  MoveL 1967 to (59.09, 49.47, 12.6) mm, rotated rx 0 ry 90 rz 0 deg; joints [-9.8, 3.924, 51.005, 168.083, 55.514, -173.186]
  Set speed (120.0 mm/s)
  MoveL 1968 to (58.95, 49.36, 12.6) mm, rotated rx 0 ry 90 rz 0 deg; joints [-9.795, 3.911, 51.041, 168.092, 55.536, -173.195]
  Set speed (1000.0 mm/s)
  MoveL 1969 to (57.64, 48.99, 12.6) mm, rotated rx 0 ry 90 rz 0 deg; joints [-9.785, 3.793, 51.363, 168.132, 55.734, -173.252]
  MoveL 1970 to (53.2, 41.89, 12.6) mm, rotated rx 0 ry 90 rz 0 deg; joints [-9.389, 3.319, 52.664, 168.719, 56.5, -173.717]
  MoveL 1971 to (53.2, 41.89, 13) mm, rotated rx 0 ry 90 rz 0 deg; joints [-9.389, 3.276, 52.71, 168.719, 56.503, -173.718]
  Set speed (60.0 mm/s)
  Call Extruder(1207.537)
  MoveL 1972 to (56.95, 45.64, 13) mm, rotated rx 0 ry 90 rz 0 deg; joints [-9.584, 3.642, 51.705, 168.401, 55.898, -173.435]
  Call Extruder(1207.555)
  MoveL 1973 to (56.95, 45.51, 13) mm, rotated rx 0 ry 90 rz 0 deg; joints [-9.576, 3.64, 51.71, 168.411, 55.9, -173.441]
  Call Extruder(1207.811)
  MoveL 1974 to (58.88, 45.5, 13) mm, rotated rx 0 ry 90 rz 0 deg; joints [-9.555, 3.805, 51.26, 168.396, 55.618, -173.386]
  Call Extruder(1208.395)
  MoveL 1975 to (58.88, 41.12, 13) mm, rotated rx 0 ry 90 rz 0 deg; joints [-9.282, 3.742, 51.43, 168.74, 55.693, -173.597]
  Call Extruder(1211.736)
  MoveL 1976 to (41.12, 58.88, 13) mm, rotated rx 0 ry 90 rz 0 deg; joints [-10.592, 2.551, 54.735, 167.469, 57.91, -173.266]
  Call Extruder(1211.737)
  MoveL 1977 to (41.12, 58.88, 13) mm, rotated rx 0 ry 90 rz 0 deg; joints [-10.592, 2.551, 54.734, 167.469, 57.91, -173.266]
  Call Extruder(1212.594)
  MoveL 1978 to (41.12, 52.43, 13) mm, rotated rx 0 ry 90 rz 0 deg; joints [-10.184, 2.46, 54.992, 167.969, 58.026, -173.561]
  Call Extruder(1213.807)
  MoveL 1979 to (47.56, 58.88, 13) mm, rotated rx 0 ry 90 rz 0 deg; joints [-10.516, 3.06, 53.31, 167.432, 57.008, -173.078]
  Call Extruder(1214.455)
  MoveL 1980 to (52.43, 58.88, 13) mm, rotated rx 0 ry 90 rz 0 deg; joints [-10.46, 3.459, 52.207, 167.398, 56.314, -172.931]
  Call Extruder(1215.450)
  MoveL 1981 to (57.72, 53.59, 13) mm, rotated rx 0 ry 90 rz 0 deg; joints [-10.071, 3.826, 51.203, 167.771, 55.644, -173.027]
  Call Extruder(1215.604)
  MoveL 1982 to (58.88, 53.59, 13) mm, rotated rx 0 ry 90 rz 0 deg; joints [-10.058, 3.926, 50.931, 167.761, 55.474, -172.991]
  Call Extruder(1216.307)
  MoveL 1983 to (58.88, 58.88, 13) mm, rotated rx 0 ry 90 rz 0 deg; joints [-10.386, 4.008, 50.706, 167.345, 55.376, -172.729]
  Call Extruder(1216.308)
  MoveL 1984 to (58.88, 58.88, 13) mm, rotated rx 0 ry 90 rz 0 deg; joints [-10.386, 4.008, 50.706, 167.345, 55.376, -172.729]
  Call Extruder(1219.649)
  MoveL 1985 to (41.12, 41.12, 13) mm, rotated rx 0 ry 90 rz 0 deg; joints [-9.467, 2.31, 55.416, 168.843, 58.217, -174.07]
  Call Extruder(1220.507)
  MoveL 1986 to (41.12, 47.56, 13) mm, rotated rx 0 ry 90 rz 0 deg; joints [-9.876, 2.394, 55.178, 168.346, 58.11, -173.781]
  Call Extruder(1221.411)
  MoveL 1987 to (45.93, 42.76, 13) mm, rotated rx 0 ry 90 rz 0 deg; joints [-9.52, 2.703, 54.307, 168.694, 57.521, -173.872]
  Call Extruder(1221.446)
  MoveL 1988 to (45.93, 43.02, 13) mm, rotated rx 0 ry 90 rz 0 deg; joints [-9.536, 2.706, 54.297, 168.673, 57.516, -173.86]
  Call Extruder(1221.975)
  MoveL 1989 to (49.9, 43.02, 13) mm, rotated rx 0 ry 90 rz 0 deg; joints [-9.494, 3.023, 53.413, 168.651, 56.955, -173.754]
  Call Extruder(1222.414)
  MoveL 1990 to (53.2, 43.02, 13) mm, rotated rx 0 ry 90 rz 0 deg; joints [-9.46, 3.292, 52.667, 168.631, 56.484, -173.664]
  Call Extruder(1222.667)
  MoveL 1991 to (53.2, 41.12, 13) mm, rotated rx 0 ry 90 rz 0 deg; joints [-9.341, 3.266, 52.739, 168.779, 56.516, -173.754]
  Call Extruder(1223.422)
  MoveL 1992 to (58.88, 41.12, 13) mm, rotated rx 0 ry 90 rz 0 deg; joints [-9.282, 3.742, 51.43, 168.739, 55.693, -173.597]
  MoveL 1993 to (59.08, 41.12, 13) mm, rotated rx 0 ry 90 rz 0 deg; joints [-9.28, 3.76, 51.383, 168.738, 55.663, -173.591]
  Set speed (120.0 mm/s)
  MoveL 1994 to (52.55, 42.37, 13) mm, rotated rx 0 ry 90 rz 0 deg; joints [-9.426, 3.229, 52.84, 168.686, 56.588, -173.713]
  Set speed (1000.0 mm/s)
  MoveL 1995 to (52.48, 42.3, 13) mm, rotated rx 0 ry 90 rz 0 deg; joints [-9.422, 3.223, 52.858, 168.692, 56.599, -173.718]
  Set speed (30.0 mm/s)
  Call Extruder(1223.475)
  MoveL 1996 to (52.48, 41.9, 13) mm, rotated rx 0 ry 90 rz 0 deg; joints [-9.397, 3.217, 52.873, 168.723, 56.606, -173.737]
  Call Extruder(1223.621)
  MoveL 1997 to (52.48, 40.8, 13) mm, rotated rx 0 ry 90 rz 0 deg; joints [-9.328, 3.202, 52.914, 168.808, 56.624, -173.788]
  Call Extruder(1223.675)
  MoveL 1998 to (52.48, 40.4, 13) mm, rotated rx 0 ry 90 rz 0 deg; joints [-9.303, 3.197, 52.929, 168.839, 56.631, -173.807]
  Call Extruder(1223.709)
  MoveL 1999 to (52.88, 40.4, 13) mm, rotated rx 0 ry 90 rz 0 deg; joints [-9.299, 3.23, 52.839, 168.837, 56.573, -173.796]
  Call Extruder(1224.603)
  MoveL 2000 to (59.6, 40.4, 13) mm, rotated rx 0 ry 90 rz 0 deg; joints [-9.23, 3.794, 51.289, 168.79, 55.599, -173.611]
  Call Extruder(1225.378)
  MoveL 2001 to (59.6, 46.22, 13) mm, rotated rx 0 ry 90 rz 0 deg; joints [-9.593, 3.877, 51.062, 168.334, 55.5, -173.33]
  Call Extruder(1225.634)
  MoveL 2002 to (57.67, 46.22, 13) mm, rotated rx 0 ry 90 rz 0 deg; joints [-9.613, 3.712, 51.514, 168.349, 55.782, -173.386]
  Call Extruder(1225.914)
  MoveL 2003 to (57.67, 48.32, 13) mm, rotated rx 0 ry 90 rz 0 deg; joints [-9.744, 3.742, 51.43, 168.184, 55.746, -173.284]
  Call Extruder(1225.967)
  MoveL 2004 to (57.67, 48.72, 13) mm, rotated rx 0 ry 90 rz 0 deg; joints [-9.769, 3.748, 51.414, 168.153, 55.739, -173.265]
  Call Extruder(1226.001)
  MoveL 2005 to (58.07, 48.72, 13) mm, rotated rx 0 ry 90 rz 0 deg; joints [-9.765, 3.782, 51.321, 168.15, 55.68, -173.253]
  Call Extruder(1226.152)
  MoveL 2006 to (59.2, 48.72, 13) mm, rotated rx 0 ry 90 rz 0 deg; joints [-9.752, 3.88, 51.056, 168.141, 55.514, -173.22]
  Call Extruder(1226.205)
  MoveL 2007 to (59.6, 48.72, 13) mm, rotated rx 0 ry 90 rz 0 deg; joints [-9.748, 3.914, 50.962, 168.138, 55.456, -173.208]
  Call Extruder(1226.239)
  MoveL 2008 to (59.6, 49.12, 13) mm, rotated rx 0 ry 90 rz 0 deg; joints [-9.773, 3.92, 50.945, 168.106, 55.449, -173.188]
  Call Extruder(1226.354)
  MoveL 2009 to (59.6, 49.99, 13) mm, rotated rx 0 ry 90 rz 0 deg; joints [-9.827, 3.933, 50.91, 168.038, 55.433, -173.146]
  Call Extruder(1226.407)
  MoveL 2010 to (59.6, 50.39, 13) mm, rotated rx 0 ry 90 rz 0 deg; joints [-9.852, 3.939, 50.894, 168.007, 55.426, -173.126]
  Call Extruder(1226.442)
  MoveL 2011 to (59.2, 50.39, 13) mm, rotated rx 0 ry 90 rz 0 deg; joints [-9.856, 3.904, 50.988, 168.01, 55.485, -173.138]
  Call Extruder(1226.592)
  MoveL 2012 to (58.07, 50.38, 13) mm, rotated rx 0 ry 90 rz 0 deg; joints [-9.868, 3.807, 51.254, 168.02, 55.651, -173.173]
  Call Extruder(1226.646)
  MoveL 2013 to (57.67, 50.38, 13) mm, rotated rx 0 ry 90 rz 0 deg; joints [-9.872, 3.772, 51.348, 168.023, 55.709, -173.185]
  Call Extruder(1226.680)
  MoveL 2014 to (57.67, 50.78, 13) mm, rotated rx 0 ry 90 rz 0 deg; joints [-9.897, 3.778, 51.331, 167.992, 55.702, -173.165]
  Call Extruder(1226.958)
  MoveL 2015 to (57.67, 52.87, 13) mm, rotated rx 0 ry 90 rz 0 deg; joints [-10.027, 3.81, 51.246, 167.828, 55.665, -173.063]
  Call Extruder(1227.215)
  MoveL 2016 to (59.6, 52.87, 13) mm, rotated rx 0 ry 90 rz 0 deg; joints [-10.006, 3.977, 50.791, 167.811, 55.381, -173.004]
  Call Extruder(1228.110)
  MoveL 2017 to (59.6, 59.6, 13) mm, rotated rx 0 ry 90 rz 0 deg; joints [-10.423, 4.083, 50.504, 167.281, 55.256, -172.67]
  Call Extruder(1230.664)
  MoveL 2018 to (40.4, 59.6, 13) mm, rotated rx 0 ry 90 rz 0 deg; joints [-10.646, 2.506, 54.862, 167.417, 57.997, -173.254]
  Call Extruder(1233.218)
  MoveL 2019 to (40.4, 40.4, 13) mm, rotated rx 0 ry 90 rz 0 deg; joints [-9.429, 2.246, 55.596, 168.902, 58.328, -174.12]
  Call Extruder(1234.050)
  MoveL 2020 to (46.65, 40.4, 13) mm, rotated rx 0 ry 90 rz 0 deg; joints [-9.363, 2.728, 54.235, 168.873, 57.458, -173.961]
  Call Extruder(1234.302)
  MoveL 2021 to (46.65, 42.3, 13) mm, rotated rx 0 ry 90 rz 0 deg; joints [-9.483, 2.753, 54.165, 168.725, 57.427, -173.874]
  Call Extruder(1234.629)
  MoveL 2022 to (49.11, 42.3, 13) mm, rotated rx 0 ry 90 rz 0 deg; joints [-9.457, 2.949, 53.619, 168.712, 57.08, -173.809]
  Call Extruder(1234.882)
  MoveL 2023 to (49.11, 40.4, 13) mm, rotated rx 0 ry 90 rz 0 deg; joints [-9.338, 2.924, 53.689, 168.859, 57.111, -173.896]
  Call Extruder(1235.009)
  MoveL 2024 to (50.06, 40.4, 13) mm, rotated rx 0 ry 90 rz 0 deg; joints [-9.328, 3, 53.476, 168.854, 56.976, -173.871]
  Call Extruder(1235.262)
  MoveL 2025 to (50.06, 42.3, 13) mm, rotated rx 0 ry 90 rz 0 deg; joints [-9.447, 3.026, 53.405, 168.706, 56.945, -173.783]
  Call Extruder(1235.531)
  MoveL 2026 to (52.08, 42.3, 13) mm, rotated rx 0 ry 90 rz 0 deg; joints [-9.426, 3.19, 52.949, 168.694, 56.656, -173.729]
  Call Extruder(1235.565)
  MoveL 2027 to (52.48, 42.3, 13) mm, rotated rx 0 ry 90 rz 0 deg; joints [-9.422, 3.223, 52.858, 168.692, 56.599, -173.718]
  Set speed (120.0 mm/s)
  MoveL 2028 to (52.48, 41.9, 13) mm, rotated rx 0 ry 90 rz 0 deg; joints [-9.397, 3.217, 52.873, 168.723, 56.606, -173.737]
  Set speed (1000.0 mm/s)
  MoveL 2029 to (52.58, 41.9, 13) mm, rotated rx 0 ry 90 rz 0 deg; joints [-9.396, 3.226, 52.85, 168.722, 56.591, -173.734]
  MoveL 2030 to (50.03, 42.33, 13) mm, rotated rx 0 ry 90 rz 0 deg; joints [-9.449, 3.024, 53.41, 168.704, 56.948, -173.783]
  MoveL 2031 to (49.58, 42.06, 13) mm, rotated rx 0 ry 90 rz 0 deg; joints [-9.437, 2.984, 53.521, 168.728, 57.017, -173.807]
  Set speed (30.0 mm/s)
  Call Extruder(1235.585)
  MoveL 2032 to (49.58, 42.62, 13) mm, rotated rx 0 ry 90 rz 0 deg; joints [-9.473, 2.991, 53.5, 168.684, 57.007, -173.781]
  Call Extruder(1235.645)
  MoveL 2033 to (49.58, 40.93, 13) mm, rotated rx 0 ry 90 rz 0 deg; joints [-9.366, 2.969, 53.563, 168.816, 57.036, -173.86]
  Set speed (120.0 mm/s)
  MoveL 2034 to (49.91, 40.82, 13) mm, rotated rx 0 ry 90 rz 0 deg; joints [-9.356, 2.994, 53.494, 168.822, 56.991, -173.856]
  Set speed (1000.0 mm/s)
  MoveL 2035 to (50.03, 42.33, 13) mm, rotated rx 0 ry 90 rz 0 deg; joints [-9.449, 3.024, 53.41, 168.704, 56.948, -173.783]
  MoveL 2036 to (52.51, 42.33, 13) mm, rotated rx 0 ry 90 rz 0 deg; joints [-9.423, 3.225, 52.851, 168.689, 56.595, -173.716]
  MoveL 2037 to (53.46, 42.14, 13) mm, rotated rx 0 ry 90 rz 0 deg; joints [-9.402, 3.301, 52.642, 168.697, 56.462, -173.699]
  MoveL 2038 to (53.46, 42.14, 13.4) mm, rotated rx 0 ry 90 rz 0 deg; joints [-9.402, 3.258, 52.689, 168.698, 56.465, -173.699]
  Set speed (60.0 mm/s)
  Call Extruder(1236.301)
  MoveL 2039 to (56.95, 45.64, 13.4) mm, rotated rx 0 ry 90 rz 0 deg; joints [-9.584, 3.599, 51.752, 168.401, 55.901, -173.436]
  Call Extruder(1236.350)
  MoveL 2040 to (56.95, 45.27, 13.4) mm, rotated rx 0 ry 90 rz 0 deg; joints [-9.561, 3.593, 51.766, 168.43, 55.908, -173.454]
  Call Extruder(1236.607)
  MoveL 2041 to (58.88, 45.27, 13.4) mm, rotated rx 0 ry 90 rz 0 deg; joints [-9.541, 3.758, 51.316, 168.415, 55.626, -173.398]
  Call Extruder(1237.159)
  MoveL 2042 to (58.88, 41.12, 13.4) mm, rotated rx 0 ry 90 rz 0 deg; joints [-9.282, 3.699, 51.477, 168.74, 55.697, -173.598]
  Call Extruder(1240.500)
  MoveL 2043 to (41.12, 58.88, 13.4) mm, rotated rx 0 ry 90 rz 0 deg; joints [-10.592, 2.508, 54.78, 167.47, 57.913, -173.267]
  Call Extruder(1240.500)
  MoveL 2044 to (41.12, 58.88, 13.4) mm, rotated rx 0 ry 90 rz 0 deg; joints [-10.592, 2.508, 54.779, 167.47, 57.913, -173.267]
  Call Extruder(1241.358)
  MoveL 2045 to (41.12, 52.43, 13.4) mm, rotated rx 0 ry 90 rz 0 deg; joints [-10.184, 2.417, 55.036, 167.969, 58.028, -173.562]
  Call Extruder(1242.571)
  MoveL 2046 to (47.57, 58.88, 13.4) mm, rotated rx 0 ry 90 rz 0 deg; joints [-10.516, 3.017, 53.356, 167.432, 57.011, -173.079]
  Call Extruder(1243.219)
  MoveL 2047 to (52.43, 58.88, 13.4) mm, rotated rx 0 ry 90 rz 0 deg; joints [-10.46, 3.416, 52.253, 167.398, 56.317, -172.932]
  Call Extruder(1244.171)
  MoveL 2048 to (57.5, 53.82, 13.4) mm, rotated rx 0 ry 90 rz 0 deg; joints [-10.088, 3.766, 51.294, 167.755, 55.677, -173.023]
  Call Extruder(1244.355)
  MoveL 2049 to (58.88, 53.82, 13.4) mm, rotated rx 0 ry 90 rz 0 deg; joints [-10.073, 3.886, 50.969, 167.744, 55.474, -172.981]
  Call Extruder(1245.028)
  MoveL 2050 to (58.88, 58.88, 13.4) mm, rotated rx 0 ry 90 rz 0 deg; joints [-10.386, 3.965, 50.753, 167.345, 55.38, -172.731]
  Call Extruder(1245.029)
  MoveL 2051 to (58.88, 58.88, 13.4) mm, rotated rx 0 ry 90 rz 0 deg; joints [-10.386, 3.965, 50.754, 167.345, 55.38, -172.731]
  Call Extruder(1248.370)
  MoveL 2052 to (41.12, 41.12, 13.4) mm, rotated rx 0 ry 90 rz 0 deg; joints [-9.467, 2.268, 55.46, 168.844, 58.219, -174.07]
  Call Extruder(1249.228)
  MoveL 2053 to (41.12, 47.56, 13.4) mm, rotated rx 0 ry 90 rz 0 deg; joints [-9.876, 2.351, 55.223, 168.346, 58.112, -173.782]
  Call Extruder(1250.090)
  MoveL 2054 to (45.7, 42.98, 13.4) mm, rotated rx 0 ry 90 rz 0 deg; joints [-9.536, 2.645, 54.394, 168.678, 57.551, -173.868]
  Call Extruder(1250.095)
  MoveL 2055 to (45.7, 43.02, 13.4) mm, rotated rx 0 ry 90 rz 0 deg; joints [-9.539, 2.646, 54.392, 168.675, 57.55, -173.867]
  Call Extruder(1250.624)
  MoveL 2056 to (49.68, 43.02, 13.4) mm, rotated rx 0 ry 90 rz 0 deg; joints [-9.497, 2.962, 53.509, 168.653, 56.99, -173.761]
  Call Extruder(1251.127)
  MoveL 2057 to (53.46, 43.02, 13.4) mm, rotated rx 0 ry 90 rz 0 deg; joints [-9.457, 3.27, 52.655, 168.63, 56.45, -173.658]
  Call Extruder(1251.380)
  MoveL 2058 to (53.46, 41.12, 13.4) mm, rotated rx 0 ry 90 rz 0 deg; joints [-9.338, 3.244, 52.727, 168.778, 56.482, -173.747]
  Call Extruder(1252.101)
  MoveL 2059 to (58.88, 41.12, 13.4) mm, rotated rx 0 ry 90 rz 0 deg; joints [-9.282, 3.699, 51.477, 168.74, 55.696, -173.598]
  MoveL 2060 to (59.08, 41.12, 13.4) mm, rotated rx 0 ry 90 rz 0 deg; joints [-9.28, 3.716, 51.43, 168.738, 55.667, -173.592]
  Set speed (120.0 mm/s)
  MoveL 2061 to (52.81, 42.37, 13.4) mm, rotated rx 0 ry 90 rz 0 deg; joints [-9.423, 3.208, 52.828, 168.684, 56.554, -173.707]
  Set speed (1000.0 mm/s)
  MoveL 2062 to (52.74, 42.3, 13.4) mm, rotated rx 0 ry 90 rz 0 deg; joints [-9.419, 3.201, 52.846, 168.69, 56.566, -173.712]
  Set speed (30.0 mm/s)
  Call Extruder(1252.154)
  MoveL 2063 to (52.74, 41.9, 13.4) mm, rotated rx 0 ry 90 rz 0 deg; joints [-9.394, 3.196, 52.861, 168.721, 56.572, -173.73]
  Call Extruder(1252.301)
  MoveL 2064 to (52.74, 40.8, 13.4) mm, rotated rx 0 ry 90 rz 0 deg; joints [-9.325, 3.181, 52.902, 168.807, 56.591, -173.782]
  Call Extruder(1252.354)
  MoveL 2065 to (52.74, 40.4, 13.4) mm, rotated rx 0 ry 90 rz 0 deg; joints [-9.3, 3.175, 52.917, 168.838, 56.597, -173.801]
  Call Extruder(1252.388)
  MoveL 2066 to (53.14, 40.4, 13.4) mm, rotated rx 0 ry 90 rz 0 deg; joints [-9.296, 3.208, 52.827, 168.836, 56.54, -173.79]
  Call Extruder(1253.248)
  MoveL 2067 to (59.6, 40.4, 13.4) mm, rotated rx 0 ry 90 rz 0 deg; joints [-9.23, 3.751, 51.336, 168.791, 55.603, -173.612]
  Call Extruder(1253.991)
  MoveL 2068 to (59.6, 45.98, 13.4) mm, rotated rx 0 ry 90 rz 0 deg; joints [-9.578, 3.83, 51.119, 168.353, 55.508, -173.342]
  Call Extruder(1254.248)
  MoveL 2069 to (57.67, 45.99, 13.4) mm, rotated rx 0 ry 90 rz 0 deg; joints [-9.598, 3.665, 51.57, 168.368, 55.79, -173.398]
  Call Extruder(1254.581)
  MoveL 2070 to (57.67, 48.49, 13.4) mm, rotated rx 0 ry 90 rz 0 deg; joints [-9.754, 3.701, 51.471, 168.172, 55.747, -173.277]
  Call Extruder(1254.837)
  MoveL 2071 to (59.6, 48.49, 13.4) mm, rotated rx 0 ry 90 rz 0 deg; joints [-9.734, 3.867, 51.019, 168.157, 55.464, -173.22]
  Call Extruder(1255.066)
  MoveL 2072 to (59.6, 50.21, 13.4) mm, rotated rx 0 ry 90 rz 0 deg; joints [-9.84, 3.893, 50.949, 168.022, 55.433, -173.136]
  Call Extruder(1255.119)
  MoveL 2073 to (59.6, 50.61, 13.4) mm, rotated rx 0 ry 90 rz 0 deg; joints [-9.865, 3.899, 50.932, 167.99, 55.426, -173.116]
  Call Extruder(1255.154)
  MoveL 2074 to (59.2, 50.61, 13.4) mm, rotated rx 0 ry 90 rz 0 deg; joints [-9.87, 3.864, 51.027, 167.993, 55.485, -173.129]
  Call Extruder(1255.304)
  MoveL 2075 to (58.07, 50.61, 13.4) mm, rotated rx 0 ry 90 rz 0 deg; joints [-9.882, 3.767, 51.292, 168.003, 55.651, -173.163]
  Call Extruder(1255.358)
  MoveL 2076 to (57.67, 50.61, 13.4) mm, rotated rx 0 ry 90 rz 0 deg; joints [-9.886, 3.733, 51.386, 168.006, 55.709, -173.175]
  Call Extruder(1255.392)
  MoveL 2077 to (57.67, 51.01, 13.4) mm, rotated rx 0 ry 90 rz 0 deg; joints [-9.911, 3.738, 51.37, 167.975, 55.702, -173.155]
  Call Extruder(1255.670)
  MoveL 2078 to (57.67, 53.1, 13.4) mm, rotated rx 0 ry 90 rz 0 deg; joints [-10.041, 3.77, 51.284, 167.811, 55.665, -173.053]
  Call Extruder(1255.927)
  MoveL 2079 to (59.6, 53.1, 13.4) mm, rotated rx 0 ry 90 rz 0 deg; joints [-10.02, 3.937, 50.829, 167.794, 55.381, -172.994]
  Call Extruder(1256.792)
  MoveL 2080 to (59.6, 59.6, 13.4) mm, rotated rx 0 ry 90 rz 0 deg; joints [-10.423, 4.039, 50.552, 167.282, 55.26, -172.672]
  Call Extruder(1259.347)
  MoveL 2081 to (40.4, 59.6, 13.4) mm, rotated rx 0 ry 90 rz 0 deg; joints [-10.646, 2.463, 54.906, 167.418, 57.999, -173.254]
  Call Extruder(1261.901)
  MoveL 2082 to (40.4, 40.4, 13.4) mm, rotated rx 0 ry 90 rz 0 deg; joints [-9.429, 2.204, 55.641, 168.902, 58.33, -174.12]
  Call Extruder(1262.702)
  MoveL 2083 to (46.42, 40.4, 13.4) mm, rotated rx 0 ry 90 rz 0 deg; joints [-9.366, 2.668, 54.33, 168.874, 57.493, -173.967]
  Call Extruder(1262.955)
  MoveL 2084 to (46.42, 42.3, 13.4) mm, rotated rx 0 ry 90 rz 0 deg; joints [-9.486, 2.693, 54.26, 168.727, 57.461, -173.88]
  Call Extruder(1263.282)
  MoveL 2085 to (48.88, 42.3, 13.4) mm, rotated rx 0 ry 90 rz 0 deg; joints [-9.46, 2.888, 53.715, 168.713, 57.115, -173.816]
  Call Extruder(1263.535)
  MoveL 2086 to (48.88, 40.4, 13.4) mm, rotated rx 0 ry 90 rz 0 deg; joints [-9.34, 2.863, 53.785, 168.861, 57.146, -173.903]
  Call Extruder(1263.725)
  MoveL 2087 to (50.31, 40.4, 13.4) mm, rotated rx 0 ry 90 rz 0 deg; joints [-9.325, 2.978, 53.465, 168.853, 56.943, -173.865]
  Call Extruder(1263.978)
  MoveL 2088 to (50.31, 42.3, 13.4) mm, rotated rx 0 ry 90 rz 0 deg; joints [-9.445, 3.003, 53.394, 168.705, 56.912, -173.777]
  Call Extruder(1264.248)
  MoveL 2089 to (52.34, 42.3, 13.4) mm, rotated rx 0 ry 90 rz 0 deg; joints [-9.424, 3.168, 52.937, 168.693, 56.623, -173.723]
  Call Extruder(1264.282)
  MoveL 2090 to (52.74, 42.3, 13.4) mm, rotated rx 0 ry 90 rz 0 deg; joints [-9.419, 3.201, 52.846, 168.69, 56.566, -173.712]
  Set speed (120.0 mm/s)
  MoveL 2091 to (52.74, 41.9, 13.4) mm, rotated rx 0 ry 90 rz 0 deg; joints [-9.394, 3.196, 52.861, 168.721, 56.572, -173.73]
  Set speed (1000.0 mm/s)
  MoveL 2092 to (52.84, 41.9, 13.4) mm, rotated rx 0 ry 90 rz 0 deg; joints [-9.393, 3.204, 52.838, 168.721, 56.558, -173.728]
  MoveL 2093 to (50.28, 42.33, 13.4) mm, rotated rx 0 ry 90 rz 0 deg; joints [-9.447, 3.001, 53.399, 168.703, 56.915, -173.777]
  MoveL 2094 to (49.6, 41.68, 13.4) mm, rotated rx 0 ry 90 rz 0 deg; joints [-9.413, 2.937, 53.578, 168.758, 57.024, -173.825]
  Set speed (30.0 mm/s)
  Call Extruder(1264.377)
  MoveL 2095 to (49.6, 41.11, 13.4) mm, rotated rx 0 ry 90 rz 0 deg; joints [-9.377, 2.93, 53.598, 168.802, 57.033, -173.851]
  Call Extruder(1264.444)
  MoveL 2096 to (49.88, 40.83, 13.4) mm, rotated rx 0 ry 90 rz 0 deg; joints [-9.357, 2.949, 53.546, 168.822, 56.998, -173.857]
  Set speed (120.0 mm/s)
  MoveL 2097 to (49.83, 40.78, 13.4) mm, rotated rx 0 ry 90 rz 0 deg; joints [-9.354, 2.944, 53.56, 168.826, 57.006, -173.861]
  Set speed (1000.0 mm/s)
  MoveL 2098 to (49.25, 41.9, 13.4) mm, rotated rx 0 ry 90 rz 0 deg; joints [-9.431, 2.913, 53.646, 168.742, 57.069, -173.824]
  Set speed (30.0 mm/s)
  Call Extruder(1264.508)
  MoveL 2099 to (49.94, 42.58, 13.4) mm, rotated rx 0 ry 90 rz 0 deg; joints [-9.466, 2.977, 53.468, 168.685, 56.961, -173.774]
  Set speed (120.0 mm/s)
  MoveL 2100 to (49.53, 42.74, 13.4) mm, rotated rx 0 ry 90 rz 0 deg; joints [-9.481, 2.946, 53.554, 168.676, 57.016, -173.778]
  Set speed (30.0 mm/s)
  Call Extruder(1264.534)
  MoveL 2101 to (49.25, 42.47, 13.4) mm, rotated rx 0 ry 90 rz 0 deg; joints [-9.466, 2.92, 53.625, 168.699, 57.059, -173.798]
  Set speed (120.0 mm/s)
  MoveL 2102 to (49.45, 42.87, 13.4) mm, rotated rx 0 ry 90 rz 0 deg; joints [-9.489, 2.941, 53.568, 168.666, 57.026, -173.774]
  Set speed (1000.0 mm/s)
  MoveL 2103 to (46.97, 42.43, 13.4) mm, rotated rx 0 ry 90 rz 0 deg; joints [-9.488, 2.738, 54.133, 168.714, 57.382, -173.86]
  MoveL 2104 to (41.12, 41.12, 13.4) mm, rotated rx 0 ry 90 rz 0 deg; joints [-9.467, 2.268, 55.46, 168.844, 58.219, -174.07]
  MoveL 2105 to (41.12, 41.12, 13.8) mm, rotated rx 0 ry 90 rz 0 deg; joints [-9.467, 2.225, 55.505, 168.844, 58.221, -174.071]
  Set speed (60.0 mm/s)
  Call Extruder(1267.875)
  MoveL 2106 to (58.88, 58.88, 13.8) mm, rotated rx 0 ry 90 rz 0 deg; joints [-10.386, 3.921, 50.801, 167.346, 55.384, -172.732]
  Call Extruder(1268.733)
  MoveL 2107 to (52.43, 58.88, 13.8) mm, rotated rx 0 ry 90 rz 0 deg; joints [-10.46, 3.373, 52.3, 167.399, 56.32, -172.933]
  Call Extruder(1269.643)
  MoveL 2108 to (57.27, 54.04, 13.8) mm, rotated rx 0 ry 90 rz 0 deg; joints [-10.104, 3.707, 51.385, 167.74, 55.709, -173.02]
  Call Extruder(1269.686)
  MoveL 2109 to (56.95, 54.04, 13.8) mm, rotated rx 0 ry 90 rz 0 deg; joints [-10.108, 3.679, 51.46, 167.743, 55.756, -173.03]
  Call Extruder(1270.209)
  MoveL 2110 to (56.95, 50.11, 13.8) mm, rotated rx 0 ry 90 rz 0 deg; joints [-9.863, 3.621, 51.621, 168.051, 55.827, -173.221]
  Call Extruder(1270.466)
  MoveL 2111 to (58.88, 50.11, 13.8) mm, rotated rx 0 ry 90 rz 0 deg; joints [-9.842, 3.786, 51.169, 168.036, 55.545, -173.164]
  Call Extruder(1270.617)
  MoveL 2112 to (58.88, 48.98, 13.8) mm, rotated rx 0 ry 90 rz 0 deg; joints [-9.772, 3.769, 51.216, 168.125, 55.565, -173.219]
  Call Extruder(1270.874)
  MoveL 2113 to (56.95, 48.98, 13.8) mm, rotated rx 0 ry 90 rz 0 deg; joints [-9.792, 3.604, 51.666, 168.14, 55.847, -173.276]
  Call Extruder(1271.318)
  MoveL 2114 to (56.95, 45.64, 13.8) mm, rotated rx 0 ry 90 rz 0 deg; joints [-9.584, 3.556, 51.798, 168.401, 55.905, -173.437]
  Call Extruder(1271.927)
  MoveL 2115 to (53.72, 42.4, 13.8) mm, rotated rx 0 ry 90 rz 0 deg; joints [-9.416, 3.24, 52.667, 168.677, 56.427, -173.681]
  Call Extruder(1272.097)
  MoveL 2116 to (53.72, 41.12, 13.8) mm, rotated rx 0 ry 90 rz 0 deg; joints [-9.335, 3.222, 52.715, 168.776, 56.449, -173.741]
  Call Extruder(1272.784)
  MoveL 2117 to (58.88, 41.12, 13.8) mm, rotated rx 0 ry 90 rz 0 deg; joints [-9.282, 3.656, 51.524, 168.74, 55.7, -173.599]
  Call Extruder(1272.784)
  MoveL 2118 to (58.88, 41.12, 13.8) mm, rotated rx 0 ry 90 rz 0 deg; joints [-9.282, 3.656, 51.524, 168.741, 55.7, -173.599]
  Call Extruder(1276.126)
  MoveL 2119 to (41.12, 58.88, 13.8) mm, rotated rx 0 ry 90 rz 0 deg; joints [-10.592, 2.466, 54.824, 167.47, 57.915, -173.267]
  Call Extruder(1276.983)
  MoveL 2120 to (47.56, 58.88, 13.8) mm, rotated rx 0 ry 90 rz 0 deg; joints [-10.516, 2.974, 53.402, 167.432, 57.014, -173.08]
  Call Extruder(1278.196)
  MoveL 2121 to (41.12, 52.43, 13.8) mm, rotated rx 0 ry 90 rz 0 deg; joints [-10.184, 2.375, 55.081, 167.97, 58.03, -173.562]
  Call Extruder(1278.844)
  MoveL 2122 to (41.12, 47.56, 13.8) mm, rotated rx 0 ry 90 rz 0 deg; joints [-9.876, 2.309, 55.267, 168.346, 58.114, -173.782]
  Call Extruder(1279.699)
  MoveL 2123 to (45.66, 43.02, 13.8) mm, rotated rx 0 ry 90 rz 0 deg; joints [-9.539, 2.601, 54.446, 168.675, 57.558, -173.868]
  MoveL 2124 to (45.8, 42.88, 13.8) mm, rotated rx 0 ry 90 rz 0 deg; joints [-9.529, 2.61, 54.42, 168.686, 57.541, -173.871]
  Set speed (120.0 mm/s)
  MoveL 2125 to (48.68, 42.33, 13.8) mm, rotated rx 0 ry 90 rz 0 deg; joints [-9.464, 2.83, 53.803, 168.713, 57.146, -173.82]
  Set speed (1000.0 mm/s)
  MoveL 2126 to (49.85, 41.12, 13.8) mm, rotated rx 0 ry 90 rz 0 deg; joints [-9.375, 2.907, 53.589, 168.8, 57.001, -173.845]
  Set speed (60.0 mm/s)
  Call Extruder(1279.761)
  MoveL 2127 to (49.37, 41.12, 13.8) mm, rotated rx 0 ry 90 rz 0 deg; joints [-9.38, 2.869, 53.694, 168.803, 57.067, -173.857]
  Call Extruder(1280.014)
  MoveL 2128 to (49.37, 43.02, 13.8) mm, rotated rx 0 ry 90 rz 0 deg; joints [-9.5, 2.895, 53.623, 168.655, 57.036, -173.77]
  Call Extruder(1280.533)
  MoveL 2129 to (45.48, 43.02, 13.8) mm, rotated rx 0 ry 90 rz 0 deg; joints [-9.541, 2.586, 54.487, 168.676, 57.584, -173.873]
  Call Extruder(1280.785)
  MoveL 2130 to (45.48, 41.12, 13.8) mm, rotated rx 0 ry 90 rz 0 deg; joints [-9.421, 2.561, 54.556, 168.824, 57.616, -173.959]
  Call Extruder(1281.365)
  MoveL 2131 to (41.12, 41.12, 13.8) mm, rotated rx 0 ry 90 rz 0 deg; joints [-9.467, 2.225, 55.504, 168.844, 58.221, -174.071]
  Call Extruder(1281.366)
  MoveL 2132 to (41.12, 41.12, 13.8) mm, rotated rx 0 ry 90 rz 0 deg; joints [-9.467, 2.225, 55.505, 168.844, 58.221, -174.071]
  Set speed (120.0 mm/s)
  MoveL 2133 to (46.17, 42.33, 13.8) mm, rotated rx 0 ry 90 rz 0 deg; joints [-9.49, 2.631, 54.36, 168.726, 57.499, -173.886]
  Set speed (1000.0 mm/s)
  MoveL 2134 to (53.07, 42.37, 13.8) mm, rotated rx 0 ry 90 rz 0 deg; joints [-9.42, 3.186, 52.816, 168.683, 56.521, -173.7]
  MoveL 2135 to (53, 42.3, 13.8) mm, rotated rx 0 ry 90 rz 0 deg; joints [-9.417, 3.179, 52.834, 168.689, 56.532, -173.706]
  Set speed (30.0 mm/s)
  Call Extruder(1281.419)
  MoveL 2136 to (53, 41.9, 13.8) mm, rotated rx 0 ry 90 rz 0 deg; joints [-9.392, 3.174, 52.849, 168.72, 56.539, -173.724]
  Call Extruder(1281.565)
  MoveL 2137 to (52.99, 40.8, 13.8) mm, rotated rx 0 ry 90 rz 0 deg; joints [-9.323, 3.159, 52.891, 168.806, 56.557, -173.776]
  Call Extruder(1281.618)
  MoveL 2138 to (52.99, 40.4, 13.8) mm, rotated rx 0 ry 90 rz 0 deg; joints [-9.297, 3.153, 52.906, 168.837, 56.564, -173.794]
  Call Extruder(1281.653)
  MoveL 2139 to (53.39, 40.4, 13.8) mm, rotated rx 0 ry 90 rz 0 deg; joints [-9.293, 3.186, 52.815, 168.834, 56.507, -173.784]
  Call Extruder(1282.478)
  MoveL 2140 to (59.6, 40.4, 13.8) mm, rotated rx 0 ry 90 rz 0 deg; joints [-9.23, 3.708, 51.383, 168.791, 55.607, -173.613]
  Call Extruder(1283.190)
  MoveL 2141 to (59.6, 45.75, 13.8) mm, rotated rx 0 ry 90 rz 0 deg; joints [-9.563, 3.784, 51.176, 168.373, 55.516, -173.355]
  Call Extruder(1283.446)
  MoveL 2142 to (57.67, 45.75, 13.8) mm, rotated rx 0 ry 90 rz 0 deg; joints [-9.583, 3.618, 51.627, 168.387, 55.798, -173.411]
  Call Extruder(1283.780)
  MoveL 2143 to (57.67, 48.26, 13.8) mm, rotated rx 0 ry 90 rz 0 deg; joints [-9.74, 3.655, 51.527, 168.191, 55.754, -173.29]
  Call Extruder(1284.037)
  MoveL 2144 to (59.6, 48.26, 13.8) mm, rotated rx 0 ry 90 rz 0 deg; joints [-9.719, 3.82, 51.075, 168.176, 55.472, -173.233]
  Call Extruder(1284.326)
  MoveL 2145 to (59.6, 50.43, 13.8) mm, rotated rx 0 ry 90 rz 0 deg; joints [-9.854, 3.853, 50.987, 168.005, 55.433, -173.126]
  Call Extruder(1284.379)
  MoveL 2146 to (59.6, 50.83, 13.8) mm, rotated rx 0 ry 90 rz 0 deg; joints [-9.879, 3.859, 50.971, 167.973, 55.426, -173.107]
  Call Extruder(1284.414)
  MoveL 2147 to (59.2, 50.83, 13.8) mm, rotated rx 0 ry 90 rz 0 deg; joints [-9.883, 3.824, 51.065, 167.977, 55.485, -173.119]
  Call Extruder(1284.564)
  MoveL 2148 to (58.07, 50.83, 13.8) mm, rotated rx 0 ry 90 rz 0 deg; joints [-9.896, 3.727, 51.33, 167.986, 55.651, -173.153]
  Call Extruder(1284.617)
  MoveL 2149 to (57.67, 50.83, 13.8) mm, rotated rx 0 ry 90 rz 0 deg; joints [-9.9, 3.693, 51.424, 167.989, 55.709, -173.165]
  Call Extruder(1284.652)
  MoveL 2150 to (57.67, 51.23, 13.8) mm, rotated rx 0 ry 90 rz 0 deg; joints [-9.925, 3.699, 51.407, 167.958, 55.702, -173.145]
  Call Extruder(1284.930)
  MoveL 2151 to (57.67, 53.32, 13.8) mm, rotated rx 0 ry 90 rz 0 deg; joints [-10.055, 3.73, 51.321, 167.793, 55.664, -173.043]
  Call Extruder(1285.187)
  MoveL 2152 to (59.6, 53.33, 13.8) mm, rotated rx 0 ry 90 rz 0 deg; joints [-10.034, 3.897, 50.867, 167.777, 55.381, -172.984]
  Call Extruder(1286.022)
  MoveL 2153 to (59.6, 59.6, 13.8) mm, rotated rx 0 ry 90 rz 0 deg; joints [-10.423, 3.996, 50.599, 167.283, 55.264, -172.673]
  Call Extruder(1288.576)
  MoveL 2154 to (40.4, 59.6, 13.8) mm, rotated rx 0 ry 90 rz 0 deg; joints [-10.646, 2.421, 54.951, 167.418, 58.001, -173.255]
  Call Extruder(1291.131)
  MoveL 2155 to (40.4, 40.4, 13.8) mm, rotated rx 0 ry 90 rz 0 deg; joints [-9.429, 2.162, 55.685, 168.902, 58.332, -174.121]
  Call Extruder(1291.849)
  MoveL 2156 to (45.8, 40.4, 13.8) mm, rotated rx 0 ry 90 rz 0 deg; joints [-9.372, 2.577, 54.512, 168.878, 57.583, -173.984]
  Call Extruder(1291.902)
  MoveL 2157 to (46.2, 40.4, 13.8) mm, rotated rx 0 ry 90 rz 0 deg; joints [-9.368, 2.608, 54.424, 168.876, 57.527, -173.973]
  Call Extruder(1291.937)
  MoveL 2158 to (46.2, 40.8, 13.8) mm, rotated rx 0 ry 90 rz 0 deg; joints [-9.393, 2.613, 54.41, 168.845, 57.52, -173.955]
  Call Extruder(1292.083)
  MoveL 2159 to (46.2, 41.9, 13.8) mm, rotated rx 0 ry 90 rz 0 deg; joints [-9.463, 2.628, 54.37, 168.759, 57.502, -173.905]
  Call Extruder(1292.136)
  MoveL 2160 to (46.2, 42.3, 13.8) mm, rotated rx 0 ry 90 rz 0 deg; joints [-9.488, 2.633, 54.355, 168.728, 57.496, -173.887]
  Call Extruder(1292.171)
  MoveL 2161 to (46.6, 42.3, 13.8) mm, rotated rx 0 ry 90 rz 0 deg; joints [-9.484, 2.664, 54.267, 168.726, 57.439, -173.876]
  Call Extruder(1292.444)
  MoveL 2162 to (48.65, 42.3, 13.8) mm, rotated rx 0 ry 90 rz 0 deg; joints [-9.462, 2.827, 53.811, 168.715, 57.15, -173.822]
  Call Extruder(1292.697)
  MoveL 2163 to (48.66, 40.4, 13.8) mm, rotated rx 0 ry 90 rz 0 deg; joints [-9.342, 2.803, 53.88, 168.863, 57.181, -173.909]
  Call Extruder(1292.951)
  MoveL 2164 to (50.56, 40.4, 13.8) mm, rotated rx 0 ry 90 rz 0 deg; joints [-9.323, 2.956, 53.454, 168.852, 56.911, -173.859]
  Call Extruder(1293.204)
  MoveL 2165 to (50.57, 42.3, 13.8) mm, rotated rx 0 ry 90 rz 0 deg; joints [-9.442, 2.981, 53.383, 168.704, 56.879, -173.771]
  Call Extruder(1293.474)
  MoveL 2166 to (52.6, 42.3, 13.8) mm, rotated rx 0 ry 90 rz 0 deg; joints [-9.421, 3.146, 52.925, 168.692, 56.589, -173.716]
  Call Extruder(1293.508)
  MoveL 2167 to (53, 42.3, 13.8) mm, rotated rx 0 ry 90 rz 0 deg; joints [-9.417, 3.179, 52.834, 168.689, 56.532, -173.706]
  Set speed (120.0 mm/s)
  MoveL 2168 to (53, 41.9, 13.8) mm, rotated rx 0 ry 90 rz 0 deg; joints [-9.392, 3.174, 52.849, 168.72, 56.539, -173.724]
  Set speed (1000.0 mm/s)
  MoveL 2169 to (53.8, 41.9, 13.8) mm, rotated rx 0 ry 90 rz 0 deg; joints [-9.383, 3.24, 52.667, 168.715, 56.424, -173.702]
  MoveL 2170 to (46.17, 42.33, 13.8) mm, rotated rx 0 ry 90 rz 0 deg; joints [-9.49, 2.631, 54.36, 168.726, 57.499, -173.886]
  MoveL 2171 to (41.12, 41.12, 13.8) mm, rotated rx 0 ry 90 rz 0 deg; joints [-9.467, 2.225, 55.505, 168.844, 58.221, -174.071]
  MoveL 2172 to (41.12, 41.12, 14.2) mm, rotated rx 0 ry 90 rz 0 deg; joints [-9.467, 2.183, 55.549, 168.844, 58.224, -174.071]
  Set speed (60.0 mm/s)
  Call Extruder(1296.850)
  MoveL 2173 to (58.88, 58.88, 14.2) mm, rotated rx 0 ry 90 rz 0 deg; joints [-10.386, 3.878, 50.849, 167.347, 55.388, -172.733]
  Call Extruder(1297.707)
  MoveL 2174 to (52.43, 58.88, 14.2) mm, rotated rx 0 ry 90 rz 0 deg; joints [-10.46, 3.33, 52.346, 167.399, 56.324, -172.934]
  Call Extruder(1298.575)
  MoveL 2175 to (57.04, 54.27, 14.2) mm, rotated rx 0 ry 90 rz 0 deg; joints [-10.121, 3.648, 51.475, 167.725, 55.742, -173.017]
  Call Extruder(1298.588)
  MoveL 2176 to (56.95, 54.27, 14.2) mm, rotated rx 0 ry 90 rz 0 deg; joints [-10.122, 3.64, 51.497, 167.726, 55.756, -173.02]
  Call Extruder(1299.112)
  MoveL 2177 to (56.95, 50.33, 14.2) mm, rotated rx 0 ry 90 rz 0 deg; joints [-9.877, 3.581, 51.659, 168.034, 55.827, -173.211]
  Call Extruder(1299.369)
  MoveL 2178 to (58.88, 50.33, 14.2) mm, rotated rx 0 ry 90 rz 0 deg; joints [-9.856, 3.746, 51.208, 168.019, 55.545, -173.154]
  Call Extruder(1299.581)
  MoveL 2179 to (58.88, 48.74, 14.2) mm, rotated rx 0 ry 90 rz 0 deg; joints [-9.757, 3.722, 51.272, 168.144, 55.573, -173.231]
  Call Extruder(1299.837)
  MoveL 2180 to (56.95, 48.74, 14.2) mm, rotated rx 0 ry 90 rz 0 deg; joints [-9.778, 3.558, 51.722, 168.159, 55.854, -173.288]
  Call Extruder(1300.250)
  MoveL 2181 to (56.95, 45.64, 14.2) mm, rotated rx 0 ry 90 rz 0 deg; joints [-9.584, 3.513, 51.845, 168.402, 55.908, -173.438]
  Call Extruder(1300.811)
  MoveL 2182 to (53.97, 42.65, 14.2) mm, rotated rx 0 ry 90 rz 0 deg; joints [-9.429, 3.221, 52.645, 168.656, 56.39, -173.663]
  Call Extruder(1301.015)
  MoveL 2183 to (53.97, 41.12, 14.2) mm, rotated rx 0 ry 90 rz 0 deg; joints [-9.333, 3.2, 52.703, 168.775, 56.415, -173.735]
  Call Extruder(1301.669)
  MoveL 2184 to (58.88, 41.12, 14.2) mm, rotated rx 0 ry 90 rz 0 deg; joints [-9.282, 3.613, 51.571, 168.741, 55.704, -173.6]
  Call Extruder(1301.669)
  MoveL 2185 to (58.88, 41.12, 14.2) mm, rotated rx 0 ry 90 rz 0 deg; joints [-9.282, 3.613, 51.571, 168.741, 55.704, -173.6]
  Call Extruder(1305.010)
  MoveL 2186 to (41.12, 58.88, 14.2) mm, rotated rx 0 ry 90 rz 0 deg; joints [-10.592, 2.424, 54.869, 167.47, 57.917, -173.268]
  Call Extruder(1305.868)
  MoveL 2187 to (47.56, 58.88, 14.2) mm, rotated rx 0 ry 90 rz 0 deg; joints [-10.516, 2.932, 53.448, 167.433, 57.017, -173.08]
  Call Extruder(1307.081)
  MoveL 2188 to (41.12, 52.43, 14.2) mm, rotated rx 0 ry 90 rz 0 deg; joints [-10.184, 2.333, 55.126, 167.97, 58.033, -173.563]
  Call Extruder(1307.728)
  MoveL 2189 to (41.12, 47.57, 14.2) mm, rotated rx 0 ry 90 rz 0 deg; joints [-9.876, 2.267, 55.312, 168.346, 58.116, -173.783]
  Call Extruder(1308.583)
  MoveL 2190 to (45.66, 43.02, 14.2) mm, rotated rx 0 ry 90 rz 0 deg; joints [-9.539, 2.558, 54.491, 168.676, 57.561, -173.869]
  MoveL 2191 to (45.81, 42.88, 14.2) mm, rotated rx 0 ry 90 rz 0 deg; joints [-9.529, 2.567, 54.465, 168.686, 57.544, -173.872]
  Set speed (120.0 mm/s)
  MoveL 2192 to (48.46, 42.33, 14.2) mm, rotated rx 0 ry 90 rz 0 deg; joints [-9.466, 2.769, 53.899, 168.714, 57.18, -173.827]
  Set speed (1000.0 mm/s)
  MoveL 2193 to (50.1, 41.12, 14.2) mm, rotated rx 0 ry 90 rz 0 deg; joints [-9.373, 2.885, 53.577, 168.799, 56.968, -173.839]
  Set speed (60.0 mm/s)
  Call Extruder(1308.710)
  MoveL 2194 to (49.15, 41.12, 14.2) mm, rotated rx 0 ry 90 rz 0 deg; joints [-9.383, 2.809, 53.789, 168.804, 57.102, -173.864]
  Call Extruder(1308.963)
  MoveL 2195 to (49.15, 43.02, 14.2) mm, rotated rx 0 ry 90 rz 0 deg; joints [-9.502, 2.834, 53.719, 168.657, 57.071, -173.777]
  Call Extruder(1309.481)
  MoveL 2196 to (45.25, 43.02, 14.2) mm, rotated rx 0 ry 90 rz 0 deg; joints [-9.544, 2.526, 54.581, 168.678, 57.618, -173.88]
  Call Extruder(1309.734)
  MoveL 2197 to (45.25, 41.12, 14.2) mm, rotated rx 0 ry 90 rz 0 deg; joints [-9.423, 2.501, 54.65, 168.825, 57.65, -173.966]
  Call Extruder(1310.284)
  MoveL 2198 to (41.12, 41.12, 14.2) mm, rotated rx 0 ry 90 rz 0 deg; joints [-9.467, 2.183, 55.549, 168.844, 58.223, -174.071]
  Call Extruder(1310.284)
  MoveL 2199 to (41.12, 41.12, 14.2) mm, rotated rx 0 ry 90 rz 0 deg; joints [-9.467, 2.183, 55.549, 168.844, 58.224, -174.071]
  Set speed (120.0 mm/s)
  MoveL 2200 to (45.94, 42.33, 14.2) mm, rotated rx 0 ry 90 rz 0 deg; joints [-9.492, 2.571, 54.455, 168.728, 57.533, -173.893]
  Set speed (1000.0 mm/s)
  MoveL 2201 to (53.32, 42.37, 14.2) mm, rotated rx 0 ry 90 rz 0 deg; joints [-9.418, 3.164, 52.804, 168.682, 56.488, -173.694]
  MoveL 2202 to (53.25, 42.3, 14.2) mm, rotated rx 0 ry 90 rz 0 deg; joints [-9.414, 3.157, 52.822, 168.688, 56.499, -173.699]
  Set speed (30.0 mm/s)
  Call Extruder(1310.337)
  MoveL 2203 to (53.25, 41.9, 14.2) mm, rotated rx 0 ry 90 rz 0 deg; joints [-9.389, 3.152, 52.837, 168.719, 56.505, -173.718]
  Call Extruder(1310.483)
  MoveL 2204 to (53.25, 40.8, 14.2) mm, rotated rx 0 ry 90 rz 0 deg; joints [-9.32, 3.137, 52.879, 168.805, 56.524, -173.77]
  Call Extruder(1310.536)
  MoveL 2205 to (53.25, 40.4, 14.2) mm, rotated rx 0 ry 90 rz 0 deg; joints [-9.295, 3.131, 52.894, 168.836, 56.53, -173.788]
  Call Extruder(1310.571)
  MoveL 2206 to (53.65, 40.4, 14.2) mm, rotated rx 0 ry 90 rz 0 deg; joints [-9.291, 3.164, 52.803, 168.833, 56.473, -173.778]
  Call Extruder(1311.363)
  MoveL 2207 to (59.6, 40.4, 14.2) mm, rotated rx 0 ry 90 rz 0 deg; joints [-9.23, 3.664, 51.43, 168.792, 55.611, -173.614]
  Call Extruder(1312.042)
  MoveL 2208 to (59.6, 45.51, 14.2) mm, rotated rx 0 ry 90 rz 0 deg; joints [-9.548, 3.737, 51.232, 168.392, 55.524, -173.367]
  Call Extruder(1312.298)
  MoveL 2209 to (57.67, 45.51, 14.2) mm, rotated rx 0 ry 90 rz 0 deg; joints [-9.568, 3.572, 51.683, 168.407, 55.806, -173.423]
  Call Extruder(1312.580)
  MoveL 2210 to (57.67, 47.62, 14.2) mm, rotated rx 0 ry 90 rz 0 deg; joints [-9.7, 3.602, 51.599, 168.241, 55.769, -173.321]
  Call Extruder(1312.633)
  MoveL 2211 to (57.67, 48.02, 14.2) mm, rotated rx 0 ry 90 rz 0 deg; joints [-9.725, 3.608, 51.583, 168.21, 55.762, -173.302]
  Call Extruder(1312.667)
  MoveL 2212 to (58.07, 48.02, 14.2) mm, rotated rx 0 ry 90 rz 0 deg; joints [-9.721, 3.642, 51.49, 168.207, 55.703, -173.29]
  Call Extruder(1312.817)
  MoveL 2213 to (59.2, 48.02, 14.2) mm, rotated rx 0 ry 90 rz 0 deg; joints [-9.709, 3.739, 51.226, 168.198, 55.539, -173.257]
  Call Extruder(1312.870)
  MoveL 2214 to (59.6, 48.02, 14.2) mm, rotated rx 0 ry 90 rz 0 deg; joints [-9.705, 3.774, 51.132, 168.194, 55.48, -173.245]
  Call Extruder(1312.905)
  MoveL 2215 to (59.6, 48.42, 14.2) mm, rotated rx 0 ry 90 rz 0 deg; joints [-9.729, 3.78, 51.116, 168.163, 55.473, -173.226]
  Call Extruder(1313.202)
  MoveL 2216 to (59.6, 50.65, 14.2) mm, rotated rx 0 ry 90 rz 0 deg; joints [-9.868, 3.813, 51.025, 167.988, 55.433, -173.116]
  Call Extruder(1313.255)
  MoveL 2217 to (59.6, 51.05, 14.2) mm, rotated rx 0 ry 90 rz 0 deg; joints [-9.893, 3.819, 51.009, 167.956, 55.426, -173.097]
  Call Extruder(1313.290)
  MoveL 2218 to (59.2, 51.05, 14.2) mm, rotated rx 0 ry 90 rz 0 deg; joints [-9.897, 3.784, 51.103, 167.96, 55.485, -173.109]
  Call Extruder(1313.440)
  MoveL 2219 to (58.07, 51.05, 14.2) mm, rotated rx 0 ry 90 rz 0 deg; joints [-9.909, 3.687, 51.368, 167.969, 55.65, -173.143]
  Call Extruder(1313.493)
  MoveL 2220 to (57.67, 51.05, 14.2) mm, rotated rx 0 ry 90 rz 0 deg; joints [-9.914, 3.653, 51.462, 167.972, 55.709, -173.155]
  Call Extruder(1313.528)
  MoveL 2221 to (57.67, 51.45, 14.2) mm, rotated rx 0 ry 90 rz 0 deg; joints [-9.939, 3.659, 51.445, 167.941, 55.702, -173.136]
  Call Extruder(1313.807)
  MoveL 2222 to (57.67, 53.55, 14.2) mm, rotated rx 0 ry 90 rz 0 deg; joints [-10.069, 3.69, 51.359, 167.776, 55.664, -173.033]
  Call Extruder(1314.064)
  MoveL 2223 to (59.6, 53.55, 14.2) mm, rotated rx 0 ry 90 rz 0 deg; joints [-10.048, 3.857, 50.905, 167.76, 55.381, -172.974]
  Call Extruder(1314.868)
  MoveL 2224 to (59.6, 59.6, 14.2) mm, rotated rx 0 ry 90 rz 0 deg; joints [-10.423, 3.952, 50.647, 167.283, 55.269, -172.674]
  Call Extruder(1317.423)
  MoveL 2225 to (40.4, 59.6, 14.2) mm, rotated rx 0 ry 90 rz 0 deg; joints [-10.646, 2.379, 54.996, 167.418, 58.004, -173.255]
  Call Extruder(1319.977)
  MoveL 2226 to (40.4, 40.4, 14.2) mm, rotated rx 0 ry 90 rz 0 deg; joints [-9.429, 2.12, 55.729, 168.903, 58.334, -174.121]
  Call Extruder(1320.665)
  MoveL 2227 to (45.57, 40.4, 14.2) mm, rotated rx 0 ry 90 rz 0 deg; joints [-9.374, 2.517, 54.606, 168.879, 57.617, -173.99]
  Call Extruder(1320.719)
  MoveL 2228 to (45.97, 40.4, 14.2) mm, rotated rx 0 ry 90 rz 0 deg; joints [-9.37, 2.548, 54.519, 168.877, 57.561, -173.98]
  Call Extruder(1320.753)
  MoveL 2229 to (45.97, 40.8, 14.2) mm, rotated rx 0 ry 90 rz 0 deg; joints [-9.395, 2.553, 54.504, 168.846, 57.554, -173.962]
  Call Extruder(1320.899)
  MoveL 2230 to (45.97, 41.9, 14.2) mm, rotated rx 0 ry 90 rz 0 deg; joints [-9.465, 2.568, 54.464, 168.761, 57.536, -173.912]
  Call Extruder(1320.953)
  MoveL 2231 to (45.97, 42.3, 14.2) mm, rotated rx 0 ry 90 rz 0 deg; joints [-9.49, 2.573, 54.449, 168.73, 57.53, -173.893]
  Call Extruder(1320.987)
  MoveL 2232 to (46.37, 42.3, 14.2) mm, rotated rx 0 ry 90 rz 0 deg; joints [-9.486, 2.604, 54.361, 168.728, 57.474, -173.883]
  Call Extruder(1321.261)
  MoveL 2233 to (48.43, 42.3, 14.2) mm, rotated rx 0 ry 90 rz 0 deg; joints [-9.465, 2.767, 53.906, 168.717, 57.185, -173.829]
  Call Extruder(1321.513)
  MoveL 2234 to (48.43, 40.4, 14.2) mm, rotated rx 0 ry 90 rz 0 deg; joints [-9.345, 2.742, 53.976, 168.864, 57.216, -173.916]
  Call Extruder(1321.831)
  MoveL 2235 to (50.82, 40.4, 14.2) mm, rotated rx 0 ry 90 rz 0 deg; joints [-9.32, 2.933, 53.443, 168.851, 56.878, -173.853]
  Call Extruder(1322.084)
  MoveL 2236 to (50.82, 42.3, 14.2) mm, rotated rx 0 ry 90 rz 0 deg; joints [-9.439, 2.959, 53.372, 168.703, 56.846, -173.765]
  Call Extruder(1322.354)
  MoveL 2237 to (52.85, 42.3, 14.2) mm, rotated rx 0 ry 90 rz 0 deg; joints [-9.418, 3.124, 52.913, 168.69, 56.556, -173.71]
  Call Extruder(1322.389)
  MoveL 2238 to (53.25, 42.3, 14.2) mm, rotated rx 0 ry 90 rz 0 deg; joints [-9.414, 3.157, 52.822, 168.688, 56.499, -173.699]
  Set speed (120.0 mm/s)
  MoveL 2239 to (53.25, 41.9, 14.2) mm, rotated rx 0 ry 90 rz 0 deg; joints [-9.389, 3.152, 52.837, 168.719, 56.505, -173.718]
  Set speed (1000.0 mm/s)
  MoveL 2240 to (54.05, 41.9, 14.2) mm, rotated rx 0 ry 90 rz 0 deg; joints [-9.381, 3.218, 52.655, 168.714, 56.391, -173.696]
  MoveL 2241 to (45.94, 42.33, 14.2) mm, rotated rx 0 ry 90 rz 0 deg; joints [-9.492, 2.571, 54.455, 168.728, 57.533, -173.893]
  MoveL 2242 to (41.12, 41.12, 14.2) mm, rotated rx 0 ry 90 rz 0 deg; joints [-9.467, 2.183, 55.549, 168.844, 58.224, -174.071]
  MoveL 2243 to (41.12, 41.12, 14.6) mm, rotated rx 0 ry 90 rz 0 deg; joints [-9.467, 2.141, 55.593, 168.844, 58.226, -174.072]
  Set speed (60.0 mm/s)
  Call Extruder(1325.730)
  MoveL 2244 to (58.88, 58.88, 14.6) mm, rotated rx 0 ry 90 rz 0 deg; joints [-10.386, 3.835, 50.896, 167.347, 55.392, -172.734]
  Call Extruder(1326.588)
  MoveL 2245 to (52.43, 58.88, 14.6) mm, rotated rx 0 ry 90 rz 0 deg; joints [-10.46, 3.287, 52.393, 167.4, 56.327, -172.935]
  Call Extruder(1327.437)
  MoveL 2246 to (56.95, 54.36, 14.6) mm, rotated rx 0 ry 90 rz 0 deg; joints [-10.128, 3.598, 51.54, 167.719, 55.758, -173.016]
  Call Extruder(1327.944)
  MoveL 2247 to (56.95, 50.55, 14.6) mm, rotated rx 0 ry 90 rz 0 deg; joints [-9.89, 3.541, 51.696, 168.018, 55.826, -173.202]
  Call Extruder(1328.201)
  MoveL 2248 to (58.88, 50.56, 14.6) mm, rotated rx 0 ry 90 rz 0 deg; joints [-9.87, 3.706, 51.246, 168.002, 55.545, -173.144]
  Call Extruder(1328.474)
  MoveL 2249 to (58.88, 48.51, 14.6) mm, rotated rx 0 ry 90 rz 0 deg; joints [-9.742, 3.676, 51.329, 168.163, 55.581, -173.244]
  Call Extruder(1328.730)
  MoveL 2250 to (56.95, 48.51, 14.6) mm, rotated rx 0 ry 90 rz 0 deg; joints [-9.763, 3.511, 51.778, 168.178, 55.862, -173.3]
  Call Extruder(1329.112)
  MoveL 2251 to (56.95, 45.64, 14.6) mm, rotated rx 0 ry 90 rz 0 deg; joints [-9.584, 3.469, 51.892, 168.402, 55.912, -173.438]
  Call Extruder(1329.625)
  MoveL 2252 to (54.23, 42.91, 14.6) mm, rotated rx 0 ry 90 rz 0 deg; joints [-9.442, 3.203, 52.623, 168.634, 56.352, -173.645]
  Call Extruder(1329.863)
  MoveL 2253 to (54.23, 41.12, 14.6) mm, rotated rx 0 ry 90 rz 0 deg; joints [-9.33, 3.179, 52.691, 168.774, 56.382, -173.729]
  Call Extruder(1330.482)
  MoveL 2254 to (58.88, 41.12, 14.6) mm, rotated rx 0 ry 90 rz 0 deg; joints [-9.282, 3.57, 51.618, 168.741, 55.708, -173.601]
  Call Extruder(1330.483)
  MoveL 2255 to (58.88, 41.12, 14.6) mm, rotated rx 0 ry 90 rz 0 deg; joints [-9.282, 3.569, 51.618, 168.742, 55.708, -173.601]
  Call Extruder(1333.824)
  MoveL 2256 to (41.12, 58.88, 14.6) mm, rotated rx 0 ry 90 rz 0 deg; joints [-10.592, 2.381, 54.914, 167.471, 57.92, -173.269]
  Call Extruder(1334.682)
  MoveL 2257 to (47.56, 58.88, 14.6) mm, rotated rx 0 ry 90 rz 0 deg; joints [-10.516, 2.889, 53.493, 167.433, 57.02, -173.081]
  Call Extruder(1335.894)
  MoveL 2258 to (41.12, 52.43, 14.6) mm, rotated rx 0 ry 90 rz 0 deg; joints [-10.184, 2.291, 55.17, 167.97, 58.035, -173.563]
  Call Extruder(1336.542)
  MoveL 2259 to (41.12, 47.57, 14.6) mm, rotated rx 0 ry 90 rz 0 deg; joints [-9.876, 2.225, 55.356, 168.347, 58.119, -173.783]
  Call Extruder(1337.397)
  MoveL 2260 to (45.66, 43.02, 14.6) mm, rotated rx 0 ry 90 rz 0 deg; joints [-9.539, 2.516, 54.536, 168.676, 57.564, -173.869]
  MoveL 2261 to (45.8, 42.88, 14.6) mm, rotated rx 0 ry 90 rz 0 deg; joints [-9.529, 2.525, 54.51, 168.686, 57.546, -173.872]
  Set speed (120.0 mm/s)
  MoveL 2262 to (41.12, 41.12, 14.6) mm, rotated rx 0 ry 90 rz 0 deg; joints [-9.467, 2.141, 55.593, 168.844, 58.225, -174.072]
  Set speed (60.0 mm/s)
  Call Extruder(1337.917)
  MoveL 2263 to (45.03, 41.12, 14.6) mm, rotated rx 0 ry 90 rz 0 deg; joints [-9.426, 2.441, 54.745, 168.826, 57.683, -173.972]
  Call Extruder(1338.170)
  MoveL 2264 to (45.03, 43.02, 14.6) mm, rotated rx 0 ry 90 rz 0 deg; joints [-9.546, 2.466, 54.675, 168.679, 57.652, -173.886]
  Call Extruder(1338.688)
  MoveL 2265 to (48.92, 43.02, 14.6) mm, rotated rx 0 ry 90 rz 0 deg; joints [-9.505, 2.773, 53.815, 168.658, 57.106, -173.783]
  Call Extruder(1338.941)
  MoveL 2266 to (48.92, 41.12, 14.6) mm, rotated rx 0 ry 90 rz 0 deg; joints [-9.385, 2.748, 53.885, 168.806, 57.137, -173.871]
  Call Extruder(1339.131)
  MoveL 2267 to (50.35, 41.12, 14.6) mm, rotated rx 0 ry 90 rz 0 deg; joints [-9.37, 2.863, 53.567, 168.798, 56.935, -173.833]
  Set speed (120.0 mm/s)
  MoveL 2268 to (48.23, 42.33, 14.6) mm, rotated rx 0 ry 90 rz 0 deg; joints [-9.468, 2.709, 53.995, 168.716, 57.215, -173.833]
  Set speed (1000.0 mm/s)
  MoveL 2269 to (45.72, 42.33, 14.6) mm, rotated rx 0 ry 90 rz 0 deg; joints [-9.495, 2.511, 54.549, 168.729, 57.567, -173.899]
  MoveL 2270 to (41.12, 41.12, 14.6) mm, rotated rx 0 ry 90 rz 0 deg; joints [-9.467, 2.141, 55.593, 168.844, 58.225, -174.072]
  Set speed (60.0 mm/s)
  Call Extruder(1339.131)
  MoveL 2271 to (41.12, 41.12, 14.6) mm, rotated rx 0 ry 90 rz 0 deg; joints [-9.467, 2.141, 55.593, 168.844, 58.226, -174.072]
  Set speed (120.0 mm/s)
  MoveL 2272 to (45.72, 42.33, 14.6) mm, rotated rx 0 ry 90 rz 0 deg; joints [-9.495, 2.511, 54.549, 168.729, 57.567, -173.899]
  Set speed (1000.0 mm/s)
  MoveL 2273 to (53.58, 42.37, 14.6) mm, rotated rx 0 ry 90 rz 0 deg; joints [-9.415, 3.142, 52.791, 168.681, 56.454, -173.688]
  MoveL 2274 to (53.51, 42.3, 14.6) mm, rotated rx 0 ry 90 rz 0 deg; joints [-9.411, 3.136, 52.81, 168.687, 56.465, -173.693]
  Set speed (30.0 mm/s)
  Call Extruder(1339.185)
  MoveL 2275 to (53.51, 41.9, 14.6) mm, rotated rx 0 ry 90 rz 0 deg; joints [-9.386, 3.13, 52.825, 168.718, 56.472, -173.712]
  Call Extruder(1339.331)
  MoveL 2276 to (53.51, 40.8, 14.6) mm, rotated rx 0 ry 90 rz 0 deg; joints [-9.317, 3.115, 52.867, 168.803, 56.49, -173.763]
  Call Extruder(1339.384)
  MoveL 2277 to (53.51, 40.4, 14.6) mm, rotated rx 0 ry 90 rz 0 deg; joints [-9.292, 3.11, 52.881, 168.835, 56.497, -173.782]
  Call Extruder(1339.419)
  MoveL 2278 to (53.91, 40.4, 14.6) mm, rotated rx 0 ry 90 rz 0 deg; joints [-9.288, 3.143, 52.79, 168.832, 56.44, -173.771]
  Call Extruder(1340.176)
  MoveL 2279 to (59.6, 40.4, 14.6) mm, rotated rx 0 ry 90 rz 0 deg; joints [-9.23, 3.621, 51.477, 168.792, 55.614, -173.615]
  Call Extruder(1340.824)
  MoveL 2280 to (59.6, 45.27, 14.6) mm, rotated rx 0 ry 90 rz 0 deg; joints [-9.533, 3.69, 51.289, 168.411, 55.532, -173.38]
  Call Extruder(1341.080)
  MoveL 2281 to (57.67, 45.27, 14.6) mm, rotated rx 0 ry 90 rz 0 deg; joints [-9.554, 3.525, 51.739, 168.426, 55.813, -173.436]
  Call Extruder(1341.362)
  MoveL 2282 to (57.67, 47.39, 14.6) mm, rotated rx 0 ry 90 rz 0 deg; joints [-9.686, 3.556, 51.655, 168.26, 55.777, -173.333]
  Call Extruder(1341.415)
  MoveL 2283 to (57.67, 47.79, 14.6) mm, rotated rx 0 ry 90 rz 0 deg; joints [-9.711, 3.562, 51.639, 168.228, 55.77, -173.314]
  Call Extruder(1341.450)
  MoveL 2284 to (58.07, 47.79, 14.6) mm, rotated rx 0 ry 90 rz 0 deg; joints [-9.706, 3.596, 51.546, 168.225, 55.711, -173.302]
  Call Extruder(1341.600)
  MoveL 2285 to (59.2, 47.79, 14.6) mm, rotated rx 0 ry 90 rz 0 deg; joints [-9.694, 3.692, 51.283, 168.217, 55.547, -173.269]
  Call Extruder(1341.653)
  MoveL 2286 to (59.6, 47.79, 14.6) mm, rotated rx 0 ry 90 rz 0 deg; joints [-9.69, 3.727, 51.189, 168.213, 55.488, -173.257]
  Call Extruder(1341.687)
  MoveL 2287 to (59.6, 48.19, 14.6) mm, rotated rx 0 ry 90 rz 0 deg; joints [-9.715, 3.733, 51.173, 168.182, 55.481, -173.238]
  Call Extruder(1342.045)
  MoveL 2288 to (59.6, 50.88, 14.6) mm, rotated rx 0 ry 90 rz 0 deg; joints [-9.882, 3.773, 51.064, 167.971, 55.433, -173.106]
  Call Extruder(1342.045)
  MoveL 2289 to (59.6, 50.88, 14.6) mm, rotated rx 0 ry 90 rz 0 deg; joints [-9.882, 3.773, 51.064, 167.971, 55.433, -173.106]
  Call Extruder(1342.099)
  MoveL 2290 to (59.6, 51.28, 14.6) mm, rotated rx 0 ry 90 rz 0 deg; joints [-9.907, 3.779, 51.047, 167.939, 55.426, -173.087]
  Call Extruder(1342.133)
  MoveL 2291 to (59.2, 51.28, 14.6) mm, rotated rx 0 ry 90 rz 0 deg; joints [-9.911, 3.744, 51.141, 167.943, 55.485, -173.099]
  Call Extruder(1342.133)
  MoveL 2292 to (59.2, 51.28, 14.6) mm, rotated rx 0 ry 90 rz 0 deg; joints [-9.911, 3.744, 51.141, 167.943, 55.485, -173.099]
  Call Extruder(1342.283)
  MoveL 2293 to (58.07, 51.27, 14.6) mm, rotated rx 0 ry 90 rz 0 deg; joints [-9.923, 3.647, 51.406, 167.952, 55.65, -173.133]
  Call Extruder(1342.337)
  MoveL 2294 to (57.67, 51.27, 14.6) mm, rotated rx 0 ry 90 rz 0 deg; joints [-9.928, 3.613, 51.499, 167.955, 55.708, -173.145]
  Call Extruder(1342.371)
  MoveL 2295 to (57.67, 51.67, 14.6) mm, rotated rx 0 ry 90 rz 0 deg; joints [-9.952, 3.619, 51.483, 167.924, 55.701, -173.126]
  Call Extruder(1342.651)
  MoveL 2296 to (57.67, 53.78, 14.6) mm, rotated rx 0 ry 90 rz 0 deg; joints [-10.083, 3.651, 51.397, 167.759, 55.664, -173.023]
  Call Extruder(1342.908)
  MoveL 2297 to (59.6, 53.78, 14.6) mm, rotated rx 0 ry 90 rz 0 deg; joints [-10.062, 3.817, 50.943, 167.743, 55.381, -172.964]
  Call Extruder(1343.682)
  MoveL 2298 to (59.6, 59.6, 14.6) mm, rotated rx 0 ry 90 rz 0 deg; joints [-10.423, 3.909, 50.695, 167.284, 55.273, -172.675]
  Call Extruder(1346.236)
  MoveL 2299 to (40.4, 59.6, 14.6) mm, rotated rx 0 ry 90 rz 0 deg; joints [-10.646, 2.336, 55.04, 167.419, 58.006, -173.256]
  Call Extruder(1348.791)
  MoveL 2300 to (40.4, 40.4, 14.6) mm, rotated rx 0 ry 90 rz 0 deg; joints [-9.429, 2.078, 55.773, 168.903, 58.336, -174.122]
  Call Extruder(1349.449)
  MoveL 2301 to (45.35, 40.4, 14.6) mm, rotated rx 0 ry 90 rz 0 deg; joints [-9.377, 2.457, 54.701, 168.88, 57.65, -173.996]
  Call Extruder(1349.502)
  MoveL 2302 to (45.75, 40.4, 14.6) mm, rotated rx 0 ry 90 rz 0 deg; joints [-9.373, 2.488, 54.613, 168.878, 57.595, -173.986]
  Call Extruder(1349.537)
  MoveL 2303 to (45.75, 40.8, 14.6) mm, rotated rx 0 ry 90 rz 0 deg; joints [-9.398, 2.493, 54.598, 168.848, 57.588, -173.968]
  Call Extruder(1349.683)
  MoveL 2304 to (45.75, 41.9, 14.6) mm, rotated rx 0 ry 90 rz 0 deg; joints [-9.468, 2.508, 54.558, 168.762, 57.57, -173.918]
  Call Extruder(1349.737)
  MoveL 2305 to (45.75, 42.3, 14.6) mm, rotated rx 0 ry 90 rz 0 deg; joints [-9.493, 2.513, 54.544, 168.731, 57.564, -173.9]
  Call Extruder(1349.771)
  MoveL 2306 to (46.15, 42.3, 14.6) mm, rotated rx 0 ry 90 rz 0 deg; joints [-9.489, 2.544, 54.456, 168.729, 57.508, -173.889]
  Call Extruder(1350.044)
  MoveL 2307 to (48.2, 42.3, 14.6) mm, rotated rx 0 ry 90 rz 0 deg; joints [-9.467, 2.706, 54.002, 168.718, 57.219, -173.835]
  Call Extruder(1350.297)
  MoveL 2308 to (48.2, 40.4, 14.6) mm, rotated rx 0 ry 90 rz 0 deg; joints [-9.347, 2.682, 54.071, 168.866, 57.25, -173.923]
  Call Extruder(1350.679)
  MoveL 2309 to (51.07, 40.4, 14.6) mm, rotated rx 0 ry 90 rz 0 deg; joints [-9.317, 2.911, 53.432, 168.849, 56.845, -173.847]
  Call Extruder(1350.932)
  MoveL 2310 to (51.07, 42.3, 14.6) mm, rotated rx 0 ry 90 rz 0 deg; joints [-9.437, 2.937, 53.361, 168.702, 56.813, -173.759]
  Call Extruder(1351.203)
  MoveL 2311 to (53.11, 42.3, 14.6) mm, rotated rx 0 ry 90 rz 0 deg; joints [-9.416, 3.103, 52.901, 168.689, 56.523, -173.704]
  Call Extruder(1351.237)
  MoveL 2312 to (53.51, 42.3, 14.6) mm, rotated rx 0 ry 90 rz 0 deg; joints [-9.411, 3.136, 52.81, 168.687, 56.465, -173.693]
  Set speed (120.0 mm/s)
  MoveL 2313 to (53.51, 41.9, 14.6) mm, rotated rx 0 ry 90 rz 0 deg; joints [-9.386, 3.13, 52.825, 168.718, 56.472, -173.712]
  Set speed (1000.0 mm/s)
  MoveL 2314 to (54.31, 41.9, 14.6) mm, rotated rx 0 ry 90 rz 0 deg; joints [-9.378, 3.196, 52.643, 168.712, 56.357, -173.69]
  MoveL 2315 to (45.72, 42.33, 14.6) mm, rotated rx 0 ry 90 rz 0 deg; joints [-9.495, 2.511, 54.549, 168.729, 57.567, -173.899]
  MoveL 2316 to (41.12, 41.12, 14.6) mm, rotated rx 0 ry 90 rz 0 deg; joints [-9.467, 2.141, 55.593, 168.844, 58.226, -174.072]
  MoveL 2317 to (41.12, 41.12, 15) mm, rotated rx 0 ry 90 rz 0 deg; joints [-9.467, 2.099, 55.637, 168.845, 58.228, -174.072]
  Set speed (60.0 mm/s)
  Call Extruder(1354.578)
  MoveL 2318 to (58.88, 58.88, 15) mm, rotated rx 0 ry 90 rz 0 deg; joints [-10.386, 3.791, 50.944, 167.348, 55.396, -172.735]
  Call Extruder(1355.436)
  MoveL 2319 to (52.43, 58.88, 15) mm, rotated rx 0 ry 90 rz 0 deg; joints [-10.46, 3.244, 52.439, 167.4, 56.331, -172.936]
  Call Extruder(1356.286)
  MoveL 2320 to (56.95, 54.36, 15) mm, rotated rx 0 ry 90 rz 0 deg; joints [-10.128, 3.555, 51.587, 167.719, 55.762, -173.017]
  Call Extruder(1356.763)
  MoveL 2321 to (56.95, 50.78, 15) mm, rotated rx 0 ry 90 rz 0 deg; joints [-9.904, 3.501, 51.734, 168.001, 55.826, -173.192]
  Call Extruder(1357.020)
  MoveL 2322 to (58.88, 50.78, 15) mm, rotated rx 0 ry 90 rz 0 deg; joints [-9.884, 3.666, 51.284, 167.985, 55.544, -173.134]
  Call Extruder(1357.353)
  MoveL 2323 to (58.88, 48.27, 15) mm, rotated rx 0 ry 90 rz 0 deg; joints [-9.728, 3.629, 51.385, 168.182, 55.589, -173.256]
  Call Extruder(1357.609)
  MoveL 2324 to (56.95, 48.28, 15) mm, rotated rx 0 ry 90 rz 0 deg; joints [-9.749, 3.465, 51.834, 168.196, 55.869, -173.312]
  Call Extruder(1357.960)
  MoveL 2325 to (56.95, 45.64, 15) mm, rotated rx 0 ry 90 rz 0 deg; joints [-9.584, 3.427, 51.938, 168.403, 55.915, -173.439]
  Call Extruder(1358.452)
  MoveL 2326 to (54.33, 43.02, 15) mm, rotated rx 0 ry 90 rz 0 deg; joints [-9.448, 3.171, 52.64, 168.625, 56.338, -173.637]
  Call Extruder(1358.472)
  MoveL 2327 to (54.48, 43.02, 15) mm, rotated rx 0 ry 90 rz 0 deg; joints [-9.446, 3.183, 52.606, 168.624, 56.316, -173.633]
  Call Extruder(1358.725)
  MoveL 2328 to (54.48, 41.12, 15) mm, rotated rx 0 ry 90 rz 0 deg; joints [-9.327, 3.157, 52.678, 168.773, 56.348, -173.723]
  Call Extruder(1359.310)
  MoveL 2329 to (58.88, 41.12, 15) mm, rotated rx 0 ry 90 rz 0 deg; joints [-9.282, 3.526, 51.665, 168.742, 55.711, -173.601]
  Call Extruder(1359.310)
  MoveL 2330 to (58.88, 41.12, 15) mm, rotated rx 0 ry 90 rz 0 deg; joints [-9.282, 3.526, 51.665, 168.742, 55.711, -173.602]
  Call Extruder(1362.652)
  MoveL 2331 to (41.12, 58.88, 15) mm, rotated rx 0 ry 90 rz 0 deg; joints [-10.592, 2.339, 54.958, 167.471, 57.922, -173.269]
  Call Extruder(1363.509)
  MoveL 2332 to (47.57, 58.88, 15) mm, rotated rx 0 ry 90 rz 0 deg; joints [-10.516, 2.846, 53.539, 167.434, 57.022, -173.082]
  Call Extruder(1364.722)
  MoveL 2333 to (41.12, 52.43, 15) mm, rotated rx 0 ry 90 rz 0 deg; joints [-10.184, 2.248, 55.215, 167.971, 58.037, -173.564]
  Call Extruder(1365.370)
  MoveL 2334 to (41.12, 47.57, 15) mm, rotated rx 0 ry 90 rz 0 deg; joints [-9.876, 2.183, 55.401, 168.347, 58.121, -173.784]
  Call Extruder(1366.225)
  MoveL 2335 to (45.66, 43.02, 15) mm, rotated rx 0 ry 90 rz 0 deg; joints [-9.539, 2.473, 54.581, 168.676, 57.566, -173.87]
  MoveL 2336 to (45.8, 42.88, 15) mm, rotated rx 0 ry 90 rz 0 deg; joints [-9.529, 2.482, 54.555, 168.686, 57.549, -173.873]
  Set speed (120.0 mm/s)
  MoveL 2337 to (41.12, 41.12, 15) mm, rotated rx 0 ry 90 rz 0 deg; joints [-9.467, 2.099, 55.637, 168.845, 58.228, -174.072]
  Set speed (60.0 mm/s)
  Call Extruder(1366.715)
  MoveL 2338 to (44.8, 41.12, 15) mm, rotated rx 0 ry 90 rz 0 deg; joints [-9.428, 2.382, 54.839, 168.828, 57.717, -173.978]
  Call Extruder(1366.968)
  MoveL 2339 to (44.8, 43.02, 15) mm, rotated rx 0 ry 90 rz 0 deg; joints [-9.548, 2.406, 54.77, 168.681, 57.686, -173.892]
  Call Extruder(1367.486)
  MoveL 2340 to (48.7, 43.02, 15) mm, rotated rx 0 ry 90 rz 0 deg; joints [-9.507, 2.713, 53.911, 168.66, 57.14, -173.79]
  Call Extruder(1367.739)
  MoveL 2341 to (48.7, 41.12, 15) mm, rotated rx 0 ry 90 rz 0 deg; joints [-9.387, 2.688, 53.981, 168.808, 57.172, -173.877]
  Call Extruder(1367.992)
  MoveL 2342 to (50.6, 41.12, 15) mm, rotated rx 0 ry 90 rz 0 deg; joints [-9.367, 2.84, 53.555, 168.797, 56.902, -173.827]
  MoveL 2343 to (50.8, 41.12, 15) mm, rotated rx 0 ry 90 rz 0 deg; joints [-9.365, 2.856, 53.511, 168.796, 56.874, -173.822]
  Set speed (120.0 mm/s)
  MoveL 2344 to (48, 42.33, 15) mm, rotated rx 0 ry 90 rz 0 deg; joints [-9.471, 2.649, 54.09, 168.717, 57.249, -173.84]
  Set speed (1000.0 mm/s)
  MoveL 2345 to (45.49, 42.33, 15) mm, rotated rx 0 ry 90 rz 0 deg; joints [-9.497, 2.451, 54.643, 168.731, 57.601, -173.906]
  MoveL 2346 to (41.12, 41.12, 15) mm, rotated rx 0 ry 90 rz 0 deg; joints [-9.467, 2.099, 55.637, 168.845, 58.228, -174.072]
  Set speed (60.0 mm/s)
  Call Extruder(1367.993)
  MoveL 2347 to (41.12, 41.12, 15) mm, rotated rx 0 ry 90 rz 0 deg; joints [-9.467, 2.099, 55.637, 168.845, 58.228, -174.072]
  Set speed (120.0 mm/s)
  MoveL 2348 to (57.6, 51.43, 15) mm, rotated rx 0 ry 90 rz 0 deg; joints [-9.938, 3.566, 51.557, 167.944, 55.72, -173.141]
  Set speed (1000.0 mm/s)
  MoveL 2349 to (57.67, 51.5, 15) mm, rotated rx 0 ry 90 rz 0 deg; joints [-9.941, 3.573, 51.537, 167.938, 55.708, -173.135]
  Set speed (30.0 mm/s)
  Call Extruder(1368.046)
  MoveL 2350 to (57.67, 51.9, 15) mm, rotated rx 0 ry 90 rz 0 deg; joints [-9.966, 3.579, 51.521, 167.907, 55.701, -173.116]
  Call Extruder(1368.326)
  MoveL 2351 to (57.67, 54, 15) mm, rotated rx 0 ry 90 rz 0 deg; joints [-10.097, 3.611, 51.434, 167.742, 55.663, -173.013]
  Call Extruder(1368.583)
  MoveL 2352 to (59.6, 54.01, 15) mm, rotated rx 0 ry 90 rz 0 deg; joints [-10.076, 3.777, 50.981, 167.725, 55.381, -172.954]
  Call Extruder(1369.327)
  MoveL 2353 to (59.6, 59.6, 15) mm, rotated rx 0 ry 90 rz 0 deg; joints [-10.423, 3.865, 50.742, 167.285, 55.277, -172.676]
  Call Extruder(1371.882)
  MoveL 2354 to (40.4, 59.6, 15) mm, rotated rx 0 ry 90 rz 0 deg; joints [-10.646, 2.294, 55.085, 167.419, 58.008, -173.257]
  Call Extruder(1374.436)
  MoveL 2355 to (40.4, 40.4, 15) mm, rotated rx 0 ry 90 rz 0 deg; joints [-9.429, 2.036, 55.817, 168.903, 58.338, -174.122]
  Call Extruder(1375.064)
  MoveL 2356 to (45.12, 40.4, 15) mm, rotated rx 0 ry 90 rz 0 deg; joints [-9.379, 2.397, 54.795, 168.882, 57.684, -174.003]
  Call Extruder(1375.118)
  MoveL 2357 to (45.52, 40.4, 15) mm, rotated rx 0 ry 90 rz 0 deg; joints [-9.375, 2.428, 54.707, 168.88, 57.628, -173.992]
  Call Extruder(1375.152)
  MoveL 2358 to (45.52, 40.8, 15) mm, rotated rx 0 ry 90 rz 0 deg; joints [-9.4, 2.434, 54.693, 168.849, 57.622, -173.974]
  Call Extruder(1375.299)
  MoveL 2359 to (45.52, 41.9, 15) mm, rotated rx 0 ry 90 rz 0 deg; joints [-9.47, 2.448, 54.653, 168.764, 57.604, -173.924]
  Call Extruder(1375.352)
  MoveL 2360 to (45.52, 42.3, 15) mm, rotated rx 0 ry 90 rz 0 deg; joints [-9.495, 2.453, 54.638, 168.733, 57.598, -173.906]
  Call Extruder(1375.386)
  MoveL 2361 to (45.92, 42.3, 15) mm, rotated rx 0 ry 90 rz 0 deg; joints [-9.491, 2.484, 54.55, 168.731, 57.542, -173.896]
  Call Extruder(1375.660)
  MoveL 2362 to (47.98, 42.3, 15) mm, rotated rx 0 ry 90 rz 0 deg; joints [-9.469, 2.646, 54.097, 168.72, 57.254, -173.842]
  Call Extruder(1375.913)
  MoveL 2363 to (47.98, 40.4, 15) mm, rotated rx 0 ry 90 rz 0 deg; joints [-9.349, 2.621, 54.167, 168.867, 57.285, -173.929]
  Call Extruder(1376.358)
  MoveL 2364 to (51.32, 40.4, 15) mm, rotated rx 0 ry 90 rz 0 deg; joints [-9.315, 2.889, 53.421, 168.848, 56.812, -173.841]
  Call Extruder(1376.611)
  MoveL 2365 to (51.32, 42.3, 15) mm, rotated rx 0 ry 90 rz 0 deg; joints [-9.434, 2.914, 53.35, 168.701, 56.78, -173.753]
  Call Extruder(1376.882)
  MoveL 2366 to (53.36, 42.3, 15) mm, rotated rx 0 ry 90 rz 0 deg; joints [-9.413, 3.081, 52.889, 168.688, 56.489, -173.698]
  Call Extruder(1376.935)
  MoveL 2367 to (53.76, 42.3, 15) mm, rotated rx 0 ry 90 rz 0 deg; joints [-9.409, 3.114, 52.798, 168.685, 56.432, -173.687]
  Call Extruder(1376.970)
  MoveL 2368 to (53.76, 41.9, 15) mm, rotated rx 0 ry 90 rz 0 deg; joints [-9.384, 3.108, 52.813, 168.716, 56.438, -173.706]
  Call Extruder(1377.116)
  MoveL 2369 to (53.76, 40.8, 15) mm, rotated rx 0 ry 90 rz 0 deg; joints [-9.315, 3.093, 52.855, 168.802, 56.457, -173.757]
  Call Extruder(1377.169)
  MoveL 2370 to (53.76, 40.4, 15) mm, rotated rx 0 ry 90 rz 0 deg; joints [-9.29, 3.088, 52.869, 168.833, 56.463, -173.776]
  Call Extruder(1377.204)
  MoveL 2371 to (54.16, 40.4, 15) mm, rotated rx 0 ry 90 rz 0 deg; joints [-9.286, 3.121, 52.778, 168.831, 56.406, -173.765]
  Call Extruder(1377.927)
  MoveL 2372 to (59.6, 40.4, 15) mm, rotated rx 0 ry 90 rz 0 deg; joints [-9.23, 3.578, 51.524, 168.793, 55.618, -173.616]
  Call Extruder(1378.543)
  MoveL 2373 to (59.6, 45.03, 15) mm, rotated rx 0 ry 90 rz 0 deg; joints [-9.518, 3.643, 51.346, 168.43, 55.54, -173.393]
  Call Extruder(1378.799)
  MoveL 2374 to (57.67, 45.03, 15) mm, rotated rx 0 ry 90 rz 0 deg; joints [-9.539, 3.479, 51.795, 168.445, 55.821, -173.448]
  Call Extruder(1379.135)
  MoveL 2375 to (57.67, 47.56, 15) mm, rotated rx 0 ry 90 rz 0 deg; joints [-9.696, 3.515, 51.695, 168.247, 55.777, -173.326]
  Call Extruder(1379.392)
  MoveL 2376 to (59.6, 47.56, 15) mm, rotated rx 0 ry 90 rz 0 deg; joints [-9.676, 3.68, 51.245, 168.232, 55.496, -173.27]
  Call Extruder(1379.863)
  MoveL 2377 to (59.6, 51.1, 15) mm, rotated rx 0 ry 90 rz 0 deg; joints [-9.896, 3.733, 51.102, 167.954, 55.433, -173.097]
  Call Extruder(1379.916)
  MoveL 2378 to (59.6, 51.5, 15) mm, rotated rx 0 ry 90 rz 0 deg; joints [-9.921, 3.739, 51.085, 167.922, 55.426, -173.077]
  Call Extruder(1379.951)
  MoveL 2379 to (59.2, 51.5, 15) mm, rotated rx 0 ry 90 rz 0 deg; joints [-9.925, 3.704, 51.179, 167.926, 55.485, -173.089]
  Call Extruder(1380.101)
  MoveL 2380 to (58.07, 51.5, 15) mm, rotated rx 0 ry 90 rz 0 deg; joints [-9.937, 3.607, 51.444, 167.935, 55.65, -173.123]
  Call Extruder(1380.136)
  MoveL 2381 to (57.67, 51.5, 15) mm, rotated rx 0 ry 90 rz 0 deg; joints [-9.941, 3.573, 51.537, 167.938, 55.708, -173.135]
  Set speed (120.0 mm/s)
  MoveL 2382 to (57.67, 51.9, 15) mm, rotated rx 0 ry 90 rz 0 deg; joints [-9.966, 3.579, 51.521, 167.907, 55.701, -173.116]
  Set speed (1000.0 mm/s)
  MoveL 2383 to (56.87, 51.9, 15) mm, rotated rx 0 ry 90 rz 0 deg; joints [-9.975, 3.511, 51.707, 167.913, 55.817, -173.14]
  MoveL 2384 to (41.12, 41.12, 15) mm, rotated rx 0 ry 90 rz 0 deg; joints [-9.467, 2.099, 55.637, 168.845, 58.228, -174.072]
  MoveL 2385 to (41.12, 41.12, 15.4) mm, rotated rx 0 ry 90 rz 0 deg; joints [-9.467, 2.057, 55.681, 168.845, 58.23, -174.073]
  Set speed (60.0 mm/s)
  Call Extruder(1383.477)
  MoveL 2386 to (58.88, 58.88, 15.4) mm, rotated rx 0 ry 90 rz 0 deg; joints [-10.386, 3.748, 50.991, 167.349, 55.4, -172.736]
  Call Extruder(1384.335)
  MoveL 2387 to (52.43, 58.88, 15.4) mm, rotated rx 0 ry 90 rz 0 deg; joints [-10.46, 3.201, 52.485, 167.401, 56.334, -172.937]
  Call Extruder(1385.184)
  MoveL 2388 to (56.95, 54.36, 15.4) mm, rotated rx 0 ry 90 rz 0 deg; joints [-10.128, 3.512, 51.634, 167.72, 55.765, -173.018]
  Call Extruder(1385.632)
  MoveL 2389 to (56.95, 51, 15.4) mm, rotated rx 0 ry 90 rz 0 deg; joints [-9.918, 3.461, 51.772, 167.984, 55.825, -173.182]
  Call Extruder(1385.888)
  MoveL 2390 to (58.88, 51, 15.4) mm, rotated rx 0 ry 90 rz 0 deg; joints [-9.897, 3.626, 51.322, 167.968, 55.544, -173.124]
  Call Extruder(1386.282)
  MoveL 2391 to (58.88, 48.04, 15.4) mm, rotated rx 0 ry 90 rz 0 deg; joints [-9.713, 3.582, 51.442, 168.2, 55.596, -173.268]
  Call Extruder(1386.538)
  MoveL 2392 to (56.96, 48.04, 15.4) mm, rotated rx 0 ry 90 rz 0 deg; joints [-9.734, 3.418, 51.889, 168.215, 55.876, -173.325]
  Call Extruder(1386.858)
  MoveL 2393 to (56.95, 45.64, 15.4) mm, rotated rx 0 ry 90 rz 0 deg; joints [-9.584, 3.384, 51.984, 168.403, 55.919, -173.44]
  Call Extruder(1387.350)
  MoveL 2394 to (54.34, 43.02, 15.4) mm, rotated rx 0 ry 90 rz 0 deg; joints [-9.448, 3.128, 52.686, 168.626, 56.341, -173.638]
  Call Extruder(1387.404)
  MoveL 2395 to (54.74, 43.02, 15.4) mm, rotated rx 0 ry 90 rz 0 deg; joints [-9.444, 3.161, 52.594, 168.623, 56.283, -173.627]
  Call Extruder(1387.657)
  MoveL 2396 to (54.74, 41.12, 15.4) mm, rotated rx 0 ry 90 rz 0 deg; joints [-9.325, 3.135, 52.666, 168.771, 56.315, -173.717]
  Call Extruder(1388.208)
  MoveL 2397 to (58.88, 41.12, 15.4) mm, rotated rx 0 ry 90 rz 0 deg; joints [-9.282, 3.483, 51.712, 168.742, 55.715, -173.602]
  Call Extruder(1388.208)
  MoveL 2398 to (58.88, 41.12, 15.4) mm, rotated rx 0 ry 90 rz 0 deg; joints [-9.282, 3.483, 51.712, 168.743, 55.715, -173.602]
  Call Extruder(1391.550)
  MoveL 2399 to (41.12, 58.88, 15.4) mm, rotated rx 0 ry 90 rz 0 deg; joints [-10.592, 2.297, 55.003, 167.471, 57.924, -173.27]
  Call Extruder(1392.407)
  MoveL 2400 to (47.57, 58.88, 15.4) mm, rotated rx 0 ry 90 rz 0 deg; joints [-10.516, 2.804, 53.584, 167.434, 57.025, -173.083]
  Call Extruder(1393.620)
  MoveL 2401 to (41.12, 52.43, 15.4) mm, rotated rx 0 ry 90 rz 0 deg; joints [-10.184, 2.206, 55.259, 167.971, 58.039, -173.564]
  Call Extruder(1394.268)
  MoveL 2402 to (41.12, 47.57, 15.4) mm, rotated rx 0 ry 90 rz 0 deg; joints [-9.876, 2.14, 55.445, 168.347, 58.123, -173.784]
  Call Extruder(1395.123)
  MoveL 2403 to (45.66, 43.02, 15.4) mm, rotated rx 0 ry 90 rz 0 deg; joints [-9.539, 2.431, 54.626, 168.677, 57.568, -173.871]
  MoveL 2404 to (45.8, 42.88, 15.4) mm, rotated rx 0 ry 90 rz 0 deg; joints [-9.529, 2.44, 54.6, 168.687, 57.551, -173.873]
  Set speed (120.0 mm/s)
  MoveL 2405 to (41.12, 41.12, 15.4) mm, rotated rx 0 ry 90 rz 0 deg; joints [-9.467, 2.057, 55.681, 168.845, 58.23, -174.073]
  Set speed (60.0 mm/s)
  Call Extruder(1395.583)
  MoveL 2406 to (44.58, 41.12, 15.4) mm, rotated rx 0 ry 90 rz 0 deg; joints [-9.43, 2.322, 54.932, 168.829, 57.751, -173.985]
  Call Extruder(1395.836)
  MoveL 2407 to (44.57, 43.02, 15.4) mm, rotated rx 0 ry 90 rz 0 deg; joints [-9.551, 2.346, 54.864, 168.682, 57.72, -173.899]
  Call Extruder(1396.354)
  MoveL 2408 to (48.47, 43.02, 15.4) mm, rotated rx 0 ry 90 rz 0 deg; joints [-9.51, 2.652, 54.006, 168.661, 57.175, -173.796]
  Call Extruder(1396.607)
  MoveL 2409 to (48.47, 41.12, 15.4) mm, rotated rx 0 ry 90 rz 0 deg; joints [-9.39, 2.627, 54.076, 168.809, 57.206, -173.884]
  Call Extruder(1396.924)
  MoveL 2410 to (50.86, 41.12, 15.4) mm, rotated rx 0 ry 90 rz 0 deg; joints [-9.365, 2.818, 53.544, 168.796, 56.869, -173.821]
  MoveL 2411 to (51.06, 41.12, 15.4) mm, rotated rx 0 ry 90 rz 0 deg; joints [-9.363, 2.834, 53.499, 168.794, 56.841, -173.816]
  Set speed (120.0 mm/s)
  MoveL 2412 to (47.78, 42.33, 15.4) mm, rotated rx 0 ry 90 rz 0 deg; joints [-9.473, 2.588, 54.185, 168.719, 57.284, -173.847]
  Set speed (1000.0 mm/s)
  MoveL 2413 to (45.27, 42.33, 15.4) mm, rotated rx 0 ry 90 rz 0 deg; joints [-9.5, 2.391, 54.738, 168.732, 57.635, -173.912]
  MoveL 2414 to (41.12, 41.12, 15.4) mm, rotated rx 0 ry 90 rz 0 deg; joints [-9.467, 2.057, 55.681, 168.845, 58.23, -174.073]
  Set speed (60.0 mm/s)
  Call Extruder(1396.924)
  MoveL 2415 to (41.12, 41.12, 15.4) mm, rotated rx 0 ry 90 rz 0 deg; joints [-9.467, 2.057, 55.681, 168.845, 58.23, -174.073]
  Set speed (120.0 mm/s)
  MoveL 2416 to (45.27, 42.33, 15.4) mm, rotated rx 0 ry 90 rz 0 deg; joints [-9.5, 2.391, 54.738, 168.732, 57.635, -173.912]
  Set speed (1000.0 mm/s)
  MoveL 2417 to (54.09, 42.37, 15.4) mm, rotated rx 0 ry 90 rz 0 deg; joints [-9.41, 3.099, 52.767, 168.678, 56.387, -173.675]
  MoveL 2418 to (54.02, 42.3, 15.4) mm, rotated rx 0 ry 90 rz 0 deg; joints [-9.406, 3.092, 52.786, 168.684, 56.398, -173.681]
  Set speed (30.0 mm/s)
  Call Extruder(1396.978)
  MoveL 2419 to (54.02, 41.9, 15.4) mm, rotated rx 0 ry 90 rz 0 deg; joints [-9.381, 3.087, 52.801, 168.715, 56.405, -173.699]
  Call Extruder(1397.124)
  MoveL 2420 to (54.02, 40.8, 15.4) mm, rotated rx 0 ry 90 rz 0 deg; joints [-9.312, 3.072, 52.842, 168.801, 56.423, -173.751]
  Call Extruder(1397.177)
  MoveL 2421 to (54.02, 40.4, 15.4) mm, rotated rx 0 ry 90 rz 0 deg; joints [-9.287, 3.066, 52.857, 168.832, 56.43, -173.77]
  Call Extruder(1397.212)
  MoveL 2422 to (54.42, 40.4, 15.4) mm, rotated rx 0 ry 90 rz 0 deg; joints [-9.283, 3.099, 52.766, 168.83, 56.372, -173.759]
  Call Extruder(1397.901)
  MoveL 2423 to (59.6, 40.4, 15.4) mm, rotated rx 0 ry 90 rz 0 deg; joints [-9.23, 3.535, 51.571, 168.793, 55.622, -173.617]
  Call Extruder(1398.485)
  MoveL 2424 to (59.6, 44.79, 15.4) mm, rotated rx 0 ry 90 rz 0 deg; joints [-9.503, 3.597, 51.402, 168.45, 55.547, -173.405]
  Call Extruder(1398.688)
  MoveL 2425 to (58.07, 44.79, 15.4) mm, rotated rx 0 ry 90 rz 0 deg; joints [-9.519, 3.466, 51.758, 168.461, 55.77, -173.449]
  Call Extruder(1398.741)
  MoveL 2426 to (57.67, 44.79, 15.4) mm, rotated rx 0 ry 90 rz 0 deg; joints [-9.524, 3.432, 51.851, 168.464, 55.828, -173.46]
  Call Extruder(1398.776)
  MoveL 2427 to (57.67, 45.19, 15.4) mm, rotated rx 0 ry 90 rz 0 deg; joints [-9.549, 3.438, 51.835, 168.433, 55.822, -173.441]
  Call Extruder(1399.059)
  MoveL 2428 to (57.68, 47.32, 15.4) mm, rotated rx 0 ry 90 rz 0 deg; joints [-9.681, 3.469, 51.751, 168.266, 55.784, -173.338]
  Call Extruder(1399.315)
  MoveL 2429 to (59.6, 47.32, 15.4) mm, rotated rx 0 ry 90 rz 0 deg; joints [-9.661, 3.634, 51.302, 168.251, 55.504, -173.282]
  Call Extruder(1399.848)
  MoveL 2430 to (59.6, 51.32, 15.4) mm, rotated rx 0 ry 90 rz 0 deg; joints [-9.91, 3.693, 51.14, 167.937, 55.433, -173.087]
  Call Extruder(1399.901)
  MoveL 2431 to (59.6, 51.72, 15.4) mm, rotated rx 0 ry 90 rz 0 deg; joints [-9.934, 3.699, 51.123, 167.906, 55.426, -173.067]
  Call Extruder(1399.935)
  MoveL 2432 to (59.2, 51.72, 15.4) mm, rotated rx 0 ry 90 rz 0 deg; joints [-9.939, 3.665, 51.217, 167.909, 55.484, -173.079]
  Call Extruder(1400.085)
  MoveL 2433 to (58.07, 51.72, 15.4) mm, rotated rx 0 ry 90 rz 0 deg; joints [-9.951, 3.568, 51.482, 167.918, 55.649, -173.113]
  Call Extruder(1400.139)
  MoveL 2434 to (57.67, 51.72, 15.4) mm, rotated rx 0 ry 90 rz 0 deg; joints [-9.955, 3.533, 51.575, 167.921, 55.708, -173.125]
  Call Extruder(1400.173)
  MoveL 2435 to (57.67, 52.12, 15.4) mm, rotated rx 0 ry 90 rz 0 deg; joints [-9.98, 3.539, 51.558, 167.89, 55.701, -173.106]
  Call Extruder(1400.454)
  MoveL 2436 to (57.67, 54.23, 15.4) mm, rotated rx 0 ry 90 rz 0 deg; joints [-10.111, 3.571, 51.472, 167.724, 55.663, -173.003]
  Call Extruder(1400.711)
  MoveL 2437 to (59.6, 54.23, 15.4) mm, rotated rx 0 ry 90 rz 0 deg; joints [-10.09, 3.738, 51.019, 167.708, 55.38, -172.943]
  Call Extruder(1401.425)
  MoveL 2438 to (59.6, 59.6, 15.4) mm, rotated rx 0 ry 90 rz 0 deg; joints [-10.423, 3.822, 50.79, 167.285, 55.281, -172.677]
  Call Extruder(1403.979)
  MoveL 2439 to (40.4, 59.6, 15.4) mm, rotated rx 0 ry 90 rz 0 deg; joints [-10.646, 2.252, 55.129, 167.419, 58.01, -173.257]
  Call Extruder(1406.534)
  MoveL 2440 to (40.4, 40.4, 15.4) mm, rotated rx 0 ry 90 rz 0 deg; joints [-9.429, 1.994, 55.862, 168.903, 58.34, -174.122]
  Call Extruder(1407.132)
  MoveL 2441 to (44.9, 40.4, 15.4) mm, rotated rx 0 ry 90 rz 0 deg; joints [-9.381, 2.338, 54.888, 168.883, 57.718, -174.009]
  Call Extruder(1407.185)
  MoveL 2442 to (45.3, 40.4, 15.4) mm, rotated rx 0 ry 90 rz 0 deg; joints [-9.377, 2.369, 54.801, 168.881, 57.662, -173.999]
  Call Extruder(1407.220)
  MoveL 2443 to (45.3, 40.8, 15.4) mm, rotated rx 0 ry 90 rz 0 deg; joints [-9.403, 2.374, 54.786, 168.85, 57.656, -173.981]
  Call Extruder(1407.366)
  MoveL 2444 to (45.3, 41.9, 15.4) mm, rotated rx 0 ry 90 rz 0 deg; joints [-9.472, 2.388, 54.747, 168.765, 57.638, -173.931]
  Call Extruder(1407.420)
  MoveL 2445 to (45.3, 42.3, 15.4) mm, rotated rx 0 ry 90 rz 0 deg; joints [-9.498, 2.393, 54.732, 168.734, 57.632, -173.913]
  Call Extruder(1407.454)
  MoveL 2446 to (45.7, 42.3, 15.4) mm, rotated rx 0 ry 90 rz 0 deg; joints [-9.493, 2.424, 54.645, 168.732, 57.576, -173.902]
  Call Extruder(1407.727)
  MoveL 2447 to (47.75, 42.3, 15.4) mm, rotated rx 0 ry 90 rz 0 deg; joints [-9.472, 2.586, 54.192, 168.721, 57.288, -173.849]
  Call Extruder(1407.981)
  MoveL 2448 to (47.75, 40.4, 15.4) mm, rotated rx 0 ry 90 rz 0 deg; joints [-9.352, 2.561, 54.262, 168.869, 57.319, -173.936]
  Call Extruder(1408.489)
  MoveL 2449 to (51.57, 40.4, 15.4) mm, rotated rx 0 ry 90 rz 0 deg; joints [-9.312, 2.867, 53.41, 168.847, 56.779, -173.835]
  Call Extruder(1408.646)
  MoveL 2450 to (51.58, 41.58, 15.4) mm, rotated rx 0 ry 90 rz 0 deg; joints [-9.386, 2.882, 53.366, 168.756, 56.759, -173.78]
  Call Extruder(1408.742)
  MoveL 2451 to (51.58, 42.3, 15.4) mm, rotated rx 0 ry 90 rz 0 deg; joints [-9.432, 2.892, 53.338, 168.699, 56.747, -173.747]
  Call Extruder(1409.014)
  MoveL 2452 to (53.62, 42.3, 15.4) mm, rotated rx 0 ry 90 rz 0 deg; joints [-9.41, 3.059, 52.877, 168.687, 56.456, -173.692]
  Call Extruder(1409.048)
  MoveL 2453 to (54.02, 42.3, 15.4) mm, rotated rx 0 ry 90 rz 0 deg; joints [-9.406, 3.092, 52.786, 168.684, 56.398, -173.681]
  Set speed (120.0 mm/s)
  MoveL 2454 to (54.02, 41.9, 15.4) mm, rotated rx 0 ry 90 rz 0 deg; joints [-9.381, 3.087, 52.801, 168.715, 56.405, -173.699]
  Set speed (1000.0 mm/s)
  MoveL 2455 to (54.82, 41.9, 15.4) mm, rotated rx 0 ry 90 rz 0 deg; joints [-9.373, 3.153, 52.618, 168.71, 56.29, -173.678]
  MoveL 2456 to (45.27, 42.33, 15.4) mm, rotated rx 0 ry 90 rz 0 deg; joints [-9.5, 2.391, 54.738, 168.732, 57.635, -173.912]
  MoveL 2457 to (41.12, 41.12, 15.4) mm, rotated rx 0 ry 90 rz 0 deg; joints [-9.467, 2.057, 55.681, 168.845, 58.23, -174.073]
  MoveL 2458 to (41.12, 41.12, 15.8) mm, rotated rx 0 ry 90 rz 0 deg; joints [-9.467, 2.015, 55.726, 168.845, 58.232, -174.073]
  Set speed (60.0 mm/s)
  Call Extruder(1412.390)
  MoveL 2459 to (58.88, 58.88, 15.8) mm, rotated rx 0 ry 90 rz 0 deg; joints [-10.386, 3.704, 51.038, 167.349, 55.404, -172.737]
  Call Extruder(1413.247)
  MoveL 2460 to (52.43, 58.88, 15.8) mm, rotated rx 0 ry 90 rz 0 deg; joints [-10.46, 3.158, 52.531, 167.401, 56.337, -172.938]
  Call Extruder(1414.097)
  MoveL 2461 to (56.95, 54.36, 15.8) mm, rotated rx 0 ry 90 rz 0 deg; joints [-10.128, 3.469, 51.681, 167.72, 55.769, -173.019]
  Call Extruder(1414.515)
  MoveL 2462 to (56.95, 51.22, 15.8) mm, rotated rx 0 ry 90 rz 0 deg; joints [-9.932, 3.422, 51.809, 167.967, 55.825, -173.172]
  Call Extruder(1414.771)
  MoveL 2463 to (58.88, 51.22, 15.8) mm, rotated rx 0 ry 90 rz 0 deg; joints [-9.911, 3.586, 51.36, 167.951, 55.544, -173.114]
  Call Extruder(1415.226)
  MoveL 2464 to (58.88, 47.81, 15.8) mm, rotated rx 0 ry 90 rz 0 deg; joints [-9.699, 3.536, 51.498, 168.219, 55.604, -173.281]
  Call Extruder(1415.481)
  MoveL 2465 to (56.97, 47.81, 15.8) mm, rotated rx 0 ry 90 rz 0 deg; joints [-9.719, 3.373, 51.943, 168.234, 55.883, -173.336]
  Call Extruder(1415.641)
  MoveL 2466 to (56.95, 46.6, 15.8) mm, rotated rx 0 ry 90 rz 0 deg; joints [-9.644, 3.354, 51.993, 168.328, 55.905, -173.395]
  Call Extruder(1415.769)
  MoveL 2467 to (56.95, 45.64, 15.8) mm, rotated rx 0 ry 90 rz 0 deg; joints [-9.584, 3.34, 52.031, 168.404, 55.922, -173.441]
  Call Extruder(1416.262)
  MoveL 2468 to (54.33, 43.02, 15.8) mm, rotated rx 0 ry 90 rz 0 deg; joints [-9.448, 3.085, 52.732, 168.626, 56.344, -173.639]
  Call Extruder(1416.349)
  MoveL 2469 to (54.99, 43.02, 15.8) mm, rotated rx 0 ry 90 rz 0 deg; joints [-9.441, 3.14, 52.582, 168.622, 56.249, -173.621]
  Call Extruder(1416.603)
  MoveL 2470 to (54.99, 41.12, 15.8) mm, rotated rx 0 ry 90 rz 0 deg; joints [-9.322, 3.114, 52.654, 168.77, 56.281, -173.71]
  Call Extruder(1417.120)
  MoveL 2471 to (58.88, 41.12, 15.8) mm, rotated rx 0 ry 90 rz 0 deg; joints [-9.282, 3.44, 51.758, 168.743, 55.718, -173.603]
  Call Extruder(1417.120)
  MoveL 2472 to (58.88, 41.12, 15.8) mm, rotated rx 0 ry 90 rz 0 deg; joints [-9.282, 3.44, 51.759, 168.743, 55.718, -173.603]
  Call Extruder(1420.461)
  MoveL 2473 to (41.12, 58.88, 15.8) mm, rotated rx 0 ry 90 rz 0 deg; joints [-10.592, 2.255, 55.047, 167.472, 57.927, -173.27]
  Call Extruder(1421.319)
  MoveL 2474 to (47.56, 58.88, 15.8) mm, rotated rx 0 ry 90 rz 0 deg; joints [-10.516, 2.761, 53.629, 167.434, 57.028, -173.083]
  Call Extruder(1422.532)
  MoveL 2475 to (41.12, 52.43, 15.8) mm, rotated rx 0 ry 90 rz 0 deg; joints [-10.184, 2.164, 55.303, 167.971, 58.041, -173.565]
  Call Extruder(1423.179)
  MoveL 2476 to (41.12, 47.57, 15.8) mm, rotated rx 0 ry 90 rz 0 deg; joints [-9.876, 2.098, 55.489, 168.348, 58.125, -173.785]
  Call Extruder(1424.034)
  MoveL 2477 to (45.66, 43.02, 15.8) mm, rotated rx 0 ry 90 rz 0 deg; joints [-9.539, 2.389, 54.67, 168.677, 57.571, -173.871]
  MoveL 2478 to (45.8, 42.88, 15.8) mm, rotated rx 0 ry 90 rz 0 deg; joints [-9.529, 2.398, 54.645, 168.687, 57.553, -173.874]
  Set speed (120.0 mm/s)
  MoveL 2479 to (41.12, 41.12, 15.8) mm, rotated rx 0 ry 90 rz 0 deg; joints [-9.467, 2.015, 55.725, 168.845, 58.231, -174.073]
  Set speed (60.0 mm/s)
  Call Extruder(1424.464)
  MoveL 2480 to (44.35, 41.12, 15.8) mm, rotated rx 0 ry 90 rz 0 deg; joints [-9.433, 2.262, 55.026, 168.831, 57.785, -173.991]
  Call Extruder(1424.717)
  MoveL 2481 to (44.35, 43.02, 15.8) mm, rotated rx 0 ry 90 rz 0 deg; joints [-9.553, 2.287, 54.958, 168.683, 57.754, -173.905]
  Call Extruder(1425.236)
  MoveL 2482 to (48.24, 43.02, 15.8) mm, rotated rx 0 ry 90 rz 0 deg; joints [-9.512, 2.592, 54.101, 168.663, 57.209, -173.803]
  Call Extruder(1425.489)
  MoveL 2483 to (48.24, 41.12, 15.8) mm, rotated rx 0 ry 90 rz 0 deg; joints [-9.392, 2.567, 54.171, 168.811, 57.24, -173.89]
  Call Extruder(1425.869)
  MoveL 2484 to (51.11, 41.12, 15.8) mm, rotated rx 0 ry 90 rz 0 deg; joints [-9.362, 2.796, 53.533, 168.794, 56.836, -173.815]
  MoveL 2485 to (51.31, 41.12, 15.8) mm, rotated rx 0 ry 90 rz 0 deg; joints [-9.36, 2.812, 53.488, 168.793, 56.808, -173.81]
  Set speed (120.0 mm/s)
  MoveL 2486 to (47.55, 42.33, 15.8) mm, rotated rx 0 ry 90 rz 0 deg; joints [-9.476, 2.528, 54.28, 168.721, 57.318, -173.853]
  Set speed (1000.0 mm/s)
  MoveL 2487 to (45.04, 42.33, 15.8) mm, rotated rx 0 ry 90 rz 0 deg; joints [-9.502, 2.331, 54.832, 168.734, 57.669, -173.919]
  MoveL 2488 to (41.12, 41.12, 15.8) mm, rotated rx 0 ry 90 rz 0 deg; joints [-9.467, 2.015, 55.725, 168.845, 58.231, -174.073]
  Set speed (60.0 mm/s)
  Call Extruder(1425.870)
  MoveL 2489 to (41.12, 41.12, 15.8) mm, rotated rx 0 ry 90 rz 0 deg; joints [-9.467, 2.015, 55.726, 168.845, 58.232, -174.073]
  Set speed (120.0 mm/s)
  MoveL 2490 to (45.04, 42.33, 15.8) mm, rotated rx 0 ry 90 rz 0 deg; joints [-9.502, 2.331, 54.832, 168.734, 57.669, -173.919]
  Set speed (1000.0 mm/s)
  MoveL 2491 to (54.34, 42.37, 15.8) mm, rotated rx 0 ry 90 rz 0 deg; joints [-9.407, 3.077, 52.755, 168.677, 56.353, -173.669]
  MoveL 2492 to (54.27, 42.3, 15.8) mm, rotated rx 0 ry 90 rz 0 deg; joints [-9.404, 3.07, 52.773, 168.683, 56.365, -173.674]
  Set speed (30.0 mm/s)
  Call Extruder(1425.923)
  MoveL 2493 to (54.27, 41.9, 15.8) mm, rotated rx 0 ry 90 rz 0 deg; joints [-9.378, 3.065, 52.788, 168.714, 56.371, -173.693]
  Call Extruder(1426.069)
  MoveL 2494 to (54.27, 40.8, 15.8) mm, rotated rx 0 ry 90 rz 0 deg; joints [-9.309, 3.05, 52.83, 168.8, 56.39, -173.745]
  Call Extruder(1426.123)
  MoveL 2495 to (54.27, 40.4, 15.8) mm, rotated rx 0 ry 90 rz 0 deg; joints [-9.284, 3.044, 52.845, 168.831, 56.396, -173.764]
  Call Extruder(1426.157)
  MoveL 2496 to (54.67, 40.4, 15.8) mm, rotated rx 0 ry 90 rz 0 deg; joints [-9.28, 3.077, 52.754, 168.828, 56.339, -173.753]
  Call Extruder(1426.813)
  MoveL 2497 to (59.6, 40.4, 15.8) mm, rotated rx 0 ry 90 rz 0 deg; joints [-9.23, 3.492, 51.618, 168.794, 55.625, -173.618]
  Call Extruder(1427.365)
  MoveL 2498 to (59.6, 44.55, 15.8) mm, rotated rx 0 ry 90 rz 0 deg; joints [-9.489, 3.55, 51.458, 168.469, 55.555, -173.418]
  Call Extruder(1427.621)
  MoveL 2499 to (57.67, 44.55, 15.8) mm, rotated rx 0 ry 90 rz 0 deg; joints [-9.509, 3.386, 51.906, 168.483, 55.836, -173.473]
  Call Extruder(1427.872)
  MoveL 2500 to (57.67, 46.44, 15.8) mm, rotated rx 0 ry 90 rz 0 deg; joints [-9.627, 3.413, 51.833, 168.336, 55.804, -173.382]
  Call Extruder(1427.893)
  MoveL 2501 to (57.67, 46.6, 15.8) mm, rotated rx 0 ry 90 rz 0 deg; joints [-9.636, 3.415, 51.827, 168.324, 55.801, -173.374]
  Call Extruder(1427.958)
  MoveL 2502 to (57.68, 47.09, 15.8) mm, rotated rx 0 ry 90 rz 0 deg; joints [-9.667, 3.423, 51.806, 168.285, 55.792, -173.35]
  Call Extruder(1427.979)
  MoveL 2503 to (57.83, 47.09, 15.8) mm, rotated rx 0 ry 90 rz 0 deg; joints [-9.665, 3.436, 51.77, 168.284, 55.769, -173.346]
  Call Extruder(1428.214)
  MoveL 2504 to (59.6, 47.09, 15.8) mm, rotated rx 0 ry 90 rz 0 deg; joints [-9.646, 3.587, 51.358, 168.27, 55.511, -173.294]
  Call Extruder(1428.807)
  MoveL 2505 to (59.6, 51.54, 15.8) mm, rotated rx 0 ry 90 rz 0 deg; joints [-9.923, 3.653, 51.178, 167.92, 55.433, -173.077]
  Call Extruder(1428.860)
  MoveL 2506 to (59.6, 51.94, 15.8) mm, rotated rx 0 ry 90 rz 0 deg; joints [-9.948, 3.659, 51.161, 167.889, 55.426, -173.057]
  Call Extruder(1428.895)
  MoveL 2507 to (59.2, 51.94, 15.8) mm, rotated rx 0 ry 90 rz 0 deg; joints [-9.953, 3.625, 51.255, 167.892, 55.484, -173.069]
  Call Extruder(1429.045)
  MoveL 2508 to (58.07, 51.94, 15.8) mm, rotated rx 0 ry 90 rz 0 deg; joints [-9.965, 3.528, 51.519, 167.901, 55.649, -173.103]
  Call Extruder(1429.098)
  MoveL 2509 to (57.67, 51.94, 15.8) mm, rotated rx 0 ry 90 rz 0 deg; joints [-9.969, 3.494, 51.613, 167.905, 55.707, -173.115]
  Call Extruder(1429.132)
  MoveL 2510 to (57.67, 52.34, 15.8) mm, rotated rx 0 ry 90 rz 0 deg; joints [-9.994, 3.5, 51.596, 167.873, 55.7, -173.096]
  Call Extruder(1429.414)
  MoveL 2511 to (57.67, 54.46, 15.8) mm, rotated rx 0 ry 90 rz 0 deg; joints [-10.125, 3.532, 51.509, 167.707, 55.662, -172.993]
  Call Extruder(1429.671)
  MoveL 2512 to (59.6, 54.46, 15.8) mm, rotated rx 0 ry 90 rz 0 deg; joints [-10.104, 3.698, 51.057, 167.691, 55.38, -172.933]
  Call Extruder(1430.354)
  MoveL 2513 to (59.6, 59.6, 15.8) mm, rotated rx 0 ry 90 rz 0 deg; joints [-10.423, 3.779, 50.837, 167.286, 55.285, -172.678]
  Call Extruder(1432.909)
  MoveL 2514 to (40.4, 59.6, 15.8) mm, rotated rx 0 ry 90 rz 0 deg; joints [-10.646, 2.21, 55.174, 167.42, 58.013, -173.258]
  Call Extruder(1435.463)
  MoveL 2515 to (40.4, 40.4, 15.8) mm, rotated rx 0 ry 90 rz 0 deg; joints [-9.429, 1.952, 55.905, 168.904, 58.342, -174.123]
  Call Extruder(1436.032)
  MoveL 2516 to (44.67, 40.4, 15.8) mm, rotated rx 0 ry 90 rz 0 deg; joints [-9.384, 2.278, 54.982, 168.885, 57.752, -174.015]
  Call Extruder(1436.032)
  MoveL 2517 to (44.67, 40.4, 15.8) mm, rotated rx 0 ry 90 rz 0 deg; joints [-9.384, 2.278, 54.982, 168.885, 57.751, -174.015]
  Call Extruder(1436.085)
  MoveL 2518 to (45.07, 40.4, 15.8) mm, rotated rx 0 ry 90 rz 0 deg; joints [-9.38, 2.309, 54.895, 168.883, 57.696, -174.005]
  Call Extruder(1436.119)
  MoveL 2519 to (45.07, 40.8, 15.8) mm, rotated rx 0 ry 90 rz 0 deg; joints [-9.405, 2.314, 54.88, 168.852, 57.689, -173.987]
  Call Extruder(1436.120)
  MoveL 2520 to (45.07, 40.8, 15.8) mm, rotated rx 0 ry 90 rz 0 deg; joints [-9.405, 2.314, 54.88, 168.852, 57.689, -173.987]
  Call Extruder(1436.266)
  MoveL 2521 to (45.07, 41.9, 15.8) mm, rotated rx 0 ry 90 rz 0 deg; joints [-9.475, 2.328, 54.841, 168.767, 57.672, -173.937]
  Call Extruder(1436.319)
  MoveL 2522 to (45.07, 42.3, 15.8) mm, rotated rx 0 ry 90 rz 0 deg; joints [-9.5, 2.333, 54.826, 168.736, 57.665, -173.919]
  Call Extruder(1436.354)
  MoveL 2523 to (45.47, 42.3, 15.8) mm, rotated rx 0 ry 90 rz 0 deg; joints [-9.496, 2.364, 54.739, 168.734, 57.61, -173.909]
  Call Extruder(1436.627)
  MoveL 2524 to (47.52, 42.3, 15.8) mm, rotated rx 0 ry 90 rz 0 deg; joints [-9.474, 2.525, 54.287, 168.723, 57.322, -173.855]
  Call Extruder(1436.880)
  MoveL 2525 to (47.53, 40.4, 15.8) mm, rotated rx 0 ry 90 rz 0 deg; joints [-9.354, 2.501, 54.356, 168.87, 57.353, -173.942]
  Call Extruder(1437.452)
  MoveL 2526 to (51.83, 40.4, 15.8) mm, rotated rx 0 ry 90 rz 0 deg; joints [-9.309, 2.845, 53.398, 168.846, 56.746, -173.829]
  Call Extruder(1437.631)
  MoveL 2527 to (51.83, 41.74, 15.8) mm, rotated rx 0 ry 90 rz 0 deg; joints [-9.394, 2.863, 53.348, 168.742, 56.723, -173.767]
  Call Extruder(1437.705)
  MoveL 2528 to (51.83, 42.3, 15.8) mm, rotated rx 0 ry 90 rz 0 deg; joints [-9.429, 2.87, 53.326, 168.698, 56.714, -173.741]
  Call Extruder(1437.977)
  MoveL 2529 to (53.87, 42.3, 15.8) mm, rotated rx 0 ry 90 rz 0 deg; joints [-9.408, 3.037, 52.864, 168.685, 56.422, -173.685]
  Call Extruder(1438.011)
  MoveL 2530 to (54.27, 42.3, 15.8) mm, rotated rx 0 ry 90 rz 0 deg; joints [-9.404, 3.07, 52.773, 168.683, 56.365, -173.674]
  Set speed (120.0 mm/s)
  MoveL 2531 to (54.27, 41.9, 15.8) mm, rotated rx 0 ry 90 rz 0 deg; joints [-9.378, 3.065, 52.788, 168.714, 56.371, -173.693]
  Set speed (1000.0 mm/s)
  MoveL 2532 to (55.07, 41.9, 15.8) mm, rotated rx 0 ry 90 rz 0 deg; joints [-9.37, 3.131, 52.606, 168.709, 56.256, -173.671]
  MoveL 2533 to (45.04, 42.33, 15.8) mm, rotated rx 0 ry 90 rz 0 deg; joints [-9.502, 2.331, 54.832, 168.734, 57.669, -173.919]
  MoveL 2534 to (41.12, 41.12, 15.8) mm, rotated rx 0 ry 90 rz 0 deg; joints [-9.467, 2.015, 55.725, 168.845, 58.231, -174.073]
  MoveL 2535 to (41.12, 41.12, 16.2) mm, rotated rx 0 ry 90 rz 0 deg; joints [-9.467, 1.973, 55.769, 168.845, 58.233, -174.073]
  Set speed (60.0 mm/s)
  Call Extruder(1438.495)
  MoveL 2536 to (44.75, 41.12, 16.2) mm, rotated rx 0 ry 90 rz 0 deg; joints [-9.429, 2.251, 54.983, 168.829, 57.731, -173.981]
  Call Extruder(1438.695)
  MoveL 2537 to (44.75, 42.62, 16.2) mm, rotated rx 0 ry 90 rz 0 deg; joints [-9.524, 2.271, 54.928, 168.713, 57.706, -173.913]
  Call Extruder(1439.106)
  MoveL 2538 to (47.84, 42.62, 16.2) mm, rotated rx 0 ry 90 rz 0 deg; joints [-9.491, 2.513, 54.25, 168.697, 57.275, -173.833]
  Call Extruder(1439.106)
  MoveL 2539 to (47.84, 42.62, 16.2) mm, rotated rx 0 ry 90 rz 0 deg; joints [-9.491, 2.513, 54.25, 168.697, 57.275, -173.833]
  Call Extruder(1439.136)
  MoveL 2540 to (48.07, 42.62, 16.2) mm, rotated rx 0 ry 90 rz 0 deg; joints [-9.488, 2.53, 54.2, 168.696, 57.243, -173.827]
  Call Extruder(1439.335)
  MoveL 2541 to (48.07, 41.12, 16.2) mm, rotated rx 0 ry 90 rz 0 deg; joints [-9.394, 2.511, 54.255, 168.812, 57.267, -173.896]
  Call Extruder(1439.759)
  MoveL 2542 to (51.26, 41.12, 16.2) mm, rotated rx 0 ry 90 rz 0 deg; joints [-9.361, 2.765, 53.545, 168.794, 56.818, -173.812]
  MoveL 2543 to (51.45, 41.12, 16.2) mm, rotated rx 0 ry 90 rz 0 deg; joints [-9.359, 2.781, 53.501, 168.793, 56.789, -173.806]
  Set speed (120.0 mm/s)
  MoveL 2544 to (46.06, 42.62, 16.2) mm, rotated rx 0 ry 90 rz 0 deg; joints [-9.51, 2.372, 54.642, 168.706, 57.524, -173.879]
  Set speed (60.0 mm/s)
  Call Extruder(1440.689)
  MoveL 2545 to (41.12, 47.56, 16.2) mm, rotated rx 0 ry 90 rz 0 deg; joints [-9.876, 2.056, 55.533, 168.348, 58.127, -173.785]
  Call Extruder(1441.337)
  MoveL 2546 to (41.12, 52.43, 16.2) mm, rotated rx 0 ry 90 rz 0 deg; joints [-10.184, 2.122, 55.347, 167.971, 58.043, -173.565]
  Call Extruder(1442.550)
  MoveL 2547 to (47.56, 58.88, 16.2) mm, rotated rx 0 ry 90 rz 0 deg; joints [-10.516, 2.719, 53.675, 167.435, 57.031, -173.084]
  Call Extruder(1443.407)
  MoveL 2548 to (41.12, 58.88, 16.2) mm, rotated rx 0 ry 90 rz 0 deg; joints [-10.592, 2.213, 55.092, 167.472, 57.929, -173.271]
  Call Extruder(1446.749)
  MoveL 2549 to (58.88, 41.12, 16.2) mm, rotated rx 0 ry 90 rz 0 deg; joints [-9.282, 3.397, 51.805, 168.744, 55.722, -173.604]
  Call Extruder(1446.749)
  MoveL 2550 to (58.88, 41.12, 16.2) mm, rotated rx 0 ry 90 rz 0 deg; joints [-9.282, 3.397, 51.805, 168.743, 55.722, -173.604]
  Call Extruder(1447.319)
  MoveL 2551 to (54.59, 41.12, 16.2) mm, rotated rx 0 ry 90 rz 0 deg; joints [-9.326, 3.038, 52.791, 168.773, 56.341, -173.722]
  Call Extruder(1447.519)
  MoveL 2552 to (54.59, 42.62, 16.2) mm, rotated rx 0 ry 90 rz 0 deg; joints [-9.42, 3.058, 52.734, 168.656, 56.316, -173.651]
  Call Extruder(1447.607)
  MoveL 2553 to (53.94, 42.62, 16.2) mm, rotated rx 0 ry 90 rz 0 deg; joints [-9.427, 3.004, 52.884, 168.66, 56.411, -173.669]
  Call Extruder(1448.250)
  MoveL 2554 to (57.35, 46.04, 16.2) mm, rotated rx 0 ry 90 rz 0 deg; joints [-9.605, 3.337, 51.969, 168.37, 55.86, -173.411]
  Call Extruder(1448.463)
  MoveL 2555 to (57.35, 47.64, 16.2) mm, rotated rx 0 ry 90 rz 0 deg; joints [-9.705, 3.36, 51.906, 168.245, 55.833, -173.334]
  Call Extruder(1448.666)
  MoveL 2556 to (58.88, 47.64, 16.2) mm, rotated rx 0 ry 90 rz 0 deg; joints [-9.689, 3.49, 51.551, 168.233, 55.611, -173.29]
  Call Extruder(1449.172)
  MoveL 2557 to (58.88, 51.44, 16.2) mm, rotated rx 0 ry 90 rz 0 deg; joints [-9.925, 3.546, 51.398, 167.934, 55.544, -173.104]
  Call Extruder(1449.429)
  MoveL 2558 to (56.95, 51.44, 16.2) mm, rotated rx 0 ry 90 rz 0 deg; joints [-9.946, 3.382, 51.847, 167.95, 55.824, -173.162]
  Call Extruder(1449.817)
  MoveL 2559 to (56.95, 54.36, 16.2) mm, rotated rx 0 ry 90 rz 0 deg; joints [-10.128, 3.426, 51.727, 167.721, 55.772, -173.02]
  Call Extruder(1450.667)
  MoveL 2560 to (52.43, 58.88, 16.2) mm, rotated rx 0 ry 90 rz 0 deg; joints [-10.46, 3.115, 52.578, 167.402, 56.34, -172.938]
  Call Extruder(1451.524)
  MoveL 2561 to (58.88, 58.88, 16.2) mm, rotated rx 0 ry 90 rz 0 deg; joints [-10.386, 3.661, 51.086, 167.35, 55.408, -172.738]
  Call Extruder(1451.525)
  MoveL 2562 to (58.88, 58.88, 16.2) mm, rotated rx 0 ry 90 rz 0 deg; joints [-10.386, 3.661, 51.086, 167.35, 55.408, -172.738]
  Call Extruder(1454.866)
  MoveL 2563 to (41.12, 41.12, 16.2) mm, rotated rx 0 ry 90 rz 0 deg; joints [-9.467, 1.973, 55.77, 168.845, 58.234, -174.073]
  Call Extruder(1454.866)
  MoveL 2564 to (41.12, 41.12, 16.2) mm, rotated rx 0 ry 90 rz 0 deg; joints [-9.467, 1.973, 55.769, 168.845, 58.233, -174.073]
  Set speed (120.0 mm/s)
  MoveL 2565 to (57.6, 52.09, 16.2) mm, rotated rx 0 ry 90 rz 0 deg; joints [-9.979, 3.447, 51.669, 167.894, 55.718, -173.111]
  Set speed (1000.0 mm/s)
  MoveL 2566 to (57.67, 52.16, 16.2) mm, rotated rx 0 ry 90 rz 0 deg; joints [-9.983, 3.454, 51.65, 167.888, 55.707, -173.106]
  Set speed (30.0 mm/s)
  Call Extruder(1454.919)
  MoveL 2567 to (57.67, 52.56, 16.2) mm, rotated rx 0 ry 90 rz 0 deg; joints [-10.008, 3.46, 51.634, 167.856, 55.7, -173.086]
  Call Extruder(1455.201)
  MoveL 2568 to (57.67, 54.68, 16.2) mm, rotated rx 0 ry 90 rz 0 deg; joints [-10.139, 3.492, 51.546, 167.69, 55.661, -172.983]
  Call Extruder(1455.455)
  MoveL 2569 to (59.58, 54.69, 16.2) mm, rotated rx 0 ry 90 rz 0 deg; joints [-10.118, 3.656, 51.099, 167.674, 55.382, -172.924]
  Call Extruder(1456.056)
  MoveL 2570 to (59.6, 59.2, 16.2) mm, rotated rx 0 ry 90 rz 0 deg; joints [-10.398, 3.729, 50.902, 167.318, 55.296, -172.699]
  Call Extruder(1456.056)
  MoveL 2571 to (59.6, 59.2, 16.2) mm, rotated rx 0 ry 90 rz 0 deg; joints [-10.398, 3.729, 50.902, 167.318, 55.296, -172.699]
  Call Extruder(1456.109)
  MoveL 2572 to (59.6, 59.6, 16.2) mm, rotated rx 0 ry 90 rz 0 deg; joints [-10.423, 3.735, 50.885, 167.287, 55.289, -172.679]
  Call Extruder(1456.144)
  MoveL 2573 to (59.2, 59.6, 16.2) mm, rotated rx 0 ry 90 rz 0 deg; joints [-10.427, 3.7, 50.979, 167.29, 55.347, -172.692]
  Call Extruder(1456.144)
  MoveL 2574 to (59.2, 59.6, 16.2) mm, rotated rx 0 ry 90 rz 0 deg; joints [-10.427, 3.7, 50.979, 167.29, 55.347, -172.692]
  Call Extruder(1458.645)
  MoveL 2575 to (40.4, 59.6, 16.2) mm, rotated rx 0 ry 90 rz 0 deg; joints [-10.646, 2.168, 55.218, 167.42, 58.015, -173.258]
  Call Extruder(1461.199)
  MoveL 2576 to (40.4, 40.4, 16.2) mm, rotated rx 0 ry 90 rz 0 deg; joints [-9.429, 1.91, 55.949, 168.904, 58.344, -174.123]
  Call Extruder(1463.753)
  MoveL 2577 to (59.6, 40.4, 16.2) mm, rotated rx 0 ry 90 rz 0 deg; joints [-9.23, 3.448, 51.665, 168.794, 55.629, -173.618]
  Call Extruder(1465.265)
  MoveL 2578 to (59.6, 51.77, 16.2) mm, rotated rx 0 ry 90 rz 0 deg; joints [-9.937, 3.613, 51.216, 167.903, 55.433, -173.067]
  Call Extruder(1465.266)
  MoveL 2579 to (59.6, 51.77, 16.2) mm, rotated rx 0 ry 90 rz 0 deg; joints [-9.937, 3.613, 51.216, 167.903, 55.433, -173.067]
  Call Extruder(1465.319)
  MoveL 2580 to (59.6, 52.17, 16.2) mm, rotated rx 0 ry 90 rz 0 deg; joints [-9.962, 3.619, 51.199, 167.872, 55.425, -173.047]
  Call Extruder(1465.353)
  MoveL 2581 to (59.2, 52.17, 16.2) mm, rotated rx 0 ry 90 rz 0 deg; joints [-9.966, 3.585, 51.293, 167.875, 55.484, -173.059]
  Call Extruder(1465.353)
  MoveL 2582 to (59.2, 52.17, 16.2) mm, rotated rx 0 ry 90 rz 0 deg; joints [-9.966, 3.585, 51.293, 167.875, 55.484, -173.059]
  Call Extruder(1465.503)
  MoveL 2583 to (58.07, 52.16, 16.2) mm, rotated rx 0 ry 90 rz 0 deg; joints [-9.978, 3.488, 51.557, 167.884, 55.649, -173.094]
  Call Extruder(1465.538)
  MoveL 2584 to (57.67, 52.16, 16.2) mm, rotated rx 0 ry 90 rz 0 deg; joints [-9.983, 3.454, 51.65, 167.888, 55.707, -173.106]
  Set speed (120.0 mm/s)
  MoveL 2585 to (57.67, 52.56, 16.2) mm, rotated rx 0 ry 90 rz 0 deg; joints [-10.008, 3.46, 51.634, 167.856, 55.7, -173.086]
  Set speed (1000.0 mm/s)
  MoveL 2586 to (57.57, 52.56, 16.2) mm, rotated rx 0 ry 90 rz 0 deg; joints [-10.009, 3.451, 51.657, 167.857, 55.714, -173.089]
  MoveL 2587 to (57.66, 47.33, 16.2) mm, rotated rx 0 ry 90 rz 0 deg; joints [-9.682, 3.382, 51.847, 168.266, 55.793, -173.34]
  Set speed (30.0 mm/s)
  Call Extruder(1465.770)
  MoveL 2588 to (57.66, 45.59, 16.2) mm, rotated rx 0 ry 90 rz 0 deg; joints [-9.574, 3.357, 51.915, 168.403, 55.823, -173.424]
  Call Extruder(1465.909)
  MoveL 2589 to (57.66, 44.54, 16.2) mm, rotated rx 0 ry 90 rz 0 deg; joints [-9.508, 3.342, 51.956, 168.485, 55.841, -173.474]
  Call Extruder(1466.061)
  MoveL 2590 to (58.81, 44.54, 16.2) mm, rotated rx 0 ry 90 rz 0 deg; joints [-9.496, 3.439, 51.69, 168.476, 55.674, -173.442]
  Call Extruder(1466.432)
  MoveL 2591 to (58.81, 47.33, 16.2) mm, rotated rx 0 ry 90 rz 0 deg; joints [-9.67, 3.48, 51.58, 168.258, 55.626, -173.307]
  Call Extruder(1466.585)
  MoveL 2592 to (57.66, 47.33, 16.2) mm, rotated rx 0 ry 90 rz 0 deg; joints [-9.682, 3.382, 51.847, 168.266, 55.793, -173.34]
  Set speed (120.0 mm/s)
  MoveL 2593 to (58.45, 46.77, 16.2) mm, rotated rx 0 ry 90 rz 0 deg; joints [-9.639, 3.44, 51.687, 168.305, 55.689, -173.344]
  Set speed (30.0 mm/s)
  Call Extruder(1466.623)
  MoveL 2594 to (58.25, 46.97, 16.2) mm, rotated rx 0 ry 90 rz 0 deg; joints [-9.653, 3.426, 51.726, 168.29, 55.715, -173.341]
  Set speed (120.0 mm/s)
  MoveL 2595 to (58.02, 46.06, 16.2) mm, rotated rx 0 ry 90 rz 0 deg; joints [-9.599, 3.394, 51.813, 168.363, 55.763, -173.391]
  Set speed (30.0 mm/s)
  Call Extruder(1466.703)
  MoveL 2596 to (58.45, 45.64, 16.2) mm, rotated rx 0 ry 90 rz 0 deg; joints [-9.568, 3.424, 51.731, 168.393, 55.708, -173.399]
  Set speed (120.0 mm/s)
  MoveL 2597 to (54.28, 42.31, 16.2) mm, rotated rx 0 ry 90 rz 0 deg; joints [-9.404, 3.029, 52.817, 168.682, 56.366, -173.674]
  Set speed (30.0 mm/s)
  Call Extruder(1467.065)
  MoveL 2598 to (51.56, 42.31, 16.2) mm, rotated rx 0 ry 90 rz 0 deg; joints [-9.432, 2.806, 53.432, 168.699, 56.754, -173.748]
  Call Extruder(1467.214)
  MoveL 2599 to (51.57, 41.19, 16.2) mm, rotated rx 0 ry 90 rz 0 deg; joints [-9.362, 2.791, 53.473, 168.787, 56.773, -173.8]
  Call Extruder(1467.576)
  MoveL 2600 to (54.28, 41.19, 16.2) mm, rotated rx 0 ry 90 rz 0 deg; joints [-9.334, 3.013, 52.859, 168.77, 56.385, -173.727]
  Call Extruder(1467.725)
  MoveL 2601 to (54.28, 42.31, 16.2) mm, rotated rx 0 ry 90 rz 0 deg; joints [-9.404, 3.029, 52.817, 168.682, 56.366, -173.674]
  Set speed (120.0 mm/s)
  MoveL 2602 to (53.49, 41.55, 16.2) mm, rotated rx 0 ry 90 rz 0 deg; joints [-9.365, 2.952, 53.027, 168.747, 56.493, -173.732]
  Set speed (30.0 mm/s)
  Call Extruder(1467.801)
  MoveL 2603 to (53.08, 41.95, 16.2) mm, rotated rx 0 ry 90 rz 0 deg; joints [-9.394, 2.925, 53.103, 168.718, 56.544, -173.724]
  Set speed (120.0 mm/s)
  MoveL 2604 to (52.35, 41.55, 16.2) mm, rotated rx 0 ry 90 rz 0 deg; joints [-9.376, 2.86, 53.282, 168.754, 56.655, -173.762]
  Set speed (30.0 mm/s)
  Call Extruder(1467.877)
  MoveL 2605 to (51.95, 41.95, 16.2) mm, rotated rx 0 ry 90 rz 0 deg; joints [-9.406, 2.833, 53.358, 168.725, 56.705, -173.754]
  Set speed (120.0 mm/s)
  MoveL 2606 to (47.76, 42.31, 16.2) mm, rotated rx 0 ry 90 rz 0 deg; joints [-9.472, 2.502, 54.28, 168.721, 57.292, -173.849]
  Set speed (30.0 mm/s)
  Call Extruder(1468.236)
  MoveL 2607 to (45.06, 42.31, 16.2) mm, rotated rx 0 ry 90 rz 0 deg; joints [-9.501, 2.291, 54.872, 168.735, 57.668, -173.919]
  Call Extruder(1468.385)
  MoveL 2608 to (45.06, 41.19, 16.2) mm, rotated rx 0 ry 90 rz 0 deg; joints [-9.43, 2.276, 54.913, 168.822, 57.687, -173.97]
  Call Extruder(1468.743)
  MoveL 2609 to (47.76, 41.19, 16.2) mm, rotated rx 0 ry 90 rz 0 deg; joints [-9.401, 2.487, 54.321, 168.808, 57.31, -173.9]
  Call Extruder(1468.893)
  MoveL 2610 to (47.76, 42.31, 16.2) mm, rotated rx 0 ry 90 rz 0 deg; joints [-9.472, 2.502, 54.28, 168.721, 57.292, -173.849]
  Set speed (120.0 mm/s)
  MoveL 2611 to (46.7, 41.55, 16.2) mm, rotated rx 0 ry 90 rz 0 deg; joints [-9.435, 2.408, 54.542, 168.786, 57.453, -173.912]
  Set speed (30.0 mm/s)
  Call Extruder(1468.968)
  MoveL 2612 to (46.29, 41.95, 16.2) mm, rotated rx 0 ry 90 rz 0 deg; joints [-9.465, 2.382, 54.616, 168.757, 57.503, -173.904]
  Set speed (120.0 mm/s)
  MoveL 2613 to (45.56, 41.55, 16.2) mm, rotated rx 0 ry 90 rz 0 deg; joints [-9.447, 2.32, 54.79, 168.792, 57.611, -173.941]
  Set speed (30.0 mm/s)
  Call Extruder(1468.995)
  MoveL 2614 to (45.42, 41.69, 16.2) mm, rotated rx 0 ry 90 rz 0 deg; joints [-9.458, 2.31, 54.816, 168.781, 57.628, -173.938]
  Set speed (120.0 mm/s)
  MoveL 2615 to (41.12, 41.12, 16.2) mm, rotated rx 0 ry 90 rz 0 deg; joints [-9.467, 1.973, 55.77, 168.845, 58.234, -174.073]
  Set speed (1000.0 mm/s)
  MoveL 2616 to (41.12, 41.12, 16.6) mm, rotated rx 0 ry 90 rz 0 deg; joints [-9.467, 1.931, 55.813, 168.846, 58.235, -174.074]
  Set speed (60.0 mm/s)
  Call Extruder(1472.337)
  MoveL 2617 to (58.88, 58.88, 16.6) mm, rotated rx 0 ry 90 rz 0 deg; joints [-10.386, 3.618, 51.133, 167.35, 55.411, -172.739]
  Call Extruder(1473.194)
  MoveL 2618 to (52.43, 58.88, 16.6) mm, rotated rx 0 ry 90 rz 0 deg; joints [-10.46, 3.073, 52.624, 167.402, 56.343, -172.939]
  Call Extruder(1474.119)
  MoveL 2619 to (57.35, 53.96, 16.6) mm, rotated rx 0 ry 90 rz 0 deg; joints [-10.098, 3.41, 51.698, 167.749, 55.725, -173.028]
  Call Extruder(1474.430)
  MoveL 2620 to (57.35, 51.62, 16.6) mm, rotated rx 0 ry 90 rz 0 deg; joints [-9.953, 3.375, 51.793, 167.933, 55.766, -173.142]
  Call Extruder(1474.634)
  MoveL 2621 to (58.88, 51.62, 16.6) mm, rotated rx 0 ry 90 rz 0 deg; joints [-9.936, 3.506, 51.437, 167.921, 55.544, -173.096]
  Call Extruder(1475.174)
  MoveL 2622 to (58.88, 47.56, 16.6) mm, rotated rx 0 ry 90 rz 0 deg; joints [-9.684, 3.446, 51.601, 168.239, 55.616, -173.294]
  Call Extruder(1475.204)
  MoveL 2623 to (58.72, 47.41, 16.6) mm, rotated rx 0 ry 90 rz 0 deg; joints [-9.676, 3.43, 51.645, 168.253, 55.642, -173.306]
  Call Extruder(1475.386)
